  [53] = {x=-3E-06, y=-7.778961, rx=0.301785, ry=175.773697, rz=18.532332, fatherId=world[0]}
  [54] = {x=-4E-06, y=-7.925734, rx=0.301782, ry=175.773696, rz=18.532336, fatherId=world[0]}
  [55] = {x=-4E-06, y=-8.072507, rx=0.301779, ry=175.773696, rz=18.532339, fatherId=world[0]}
  [56] = {x=-4E-06, y=-8.21928, rx=0.301775, ry=175.773696, rz=18.532342, fatherId=world[0]}
  [57] = {x=-4E-06, y=-8.366053, rx=0.301772, ry=175.773696, rz=18.532345, fatherId=world[0]}
  [58] = {x=-4E-06, y=-8.512826, rx=0.301769, ry=175.773695, rz=18.532348, fatherId=world[0]}
  [59] = {x=-4E-06, y=-8.659599, rx=0.301766, ry=175.773695, rz=18.532352, fatherId=world[0]}
  [60] = {x=-4E-06, y=-8.806371, rx=0.301763, ry=175.773695, rz=18.532355, fatherId=world[0]}
  [61] = {x=-4E-06, y=-8.953144, rx=0.301759, ry=175.773694, rz=18.532358, fatherId=world[0]}
  [62] = {x=-4E-06, y=-9.099917, rx=0.301756, ry=175.773694, rz=18.532361, fatherId=world[0]}
  [63] = {x=-4E-06, y=-9.24669, rx=0.301753, ry=175.773694, rz=18.532364, fatherId=world[0]}
  [64] = {x=-4E-06, y=-9.393463, rx=0.30175, ry=175.773693, rz=18.532368, fatherId=world[0]}
  [65] = {x=-4E-06, y=-9.540236, rx=0.301747, ry=175.773693, rz=18.532371, fatherId=world[0]}
  [66] = {x=-4E-06, y=-9.687009, rx=0.301743, ry=175.773693, rz=18.532374, fatherId=world[0]}
  [67] = {x=-4E-06, y=-9.833781, rx=0.30174, ry=175.773693, rz=18.532377, fatherId=world[0]}
  [68] = {x=-5E-06, y=-9.980554, rx=0.301737, ry=175.773692, rz=18.53238, fatherId=world[0]}
  [69] = {x=-5E-06, y=-10.127327, rx=0.301734, ry=175.773692, rz=18.532384, fatherId=world[0]}
  [70] = {x=-5E-06, y=-10.2741, rx=0.301731, ry=175.773692, rz=18.532387, fatherId=world[0]}
  [71] = {x=-5E-06, y=-10.420873, rx=0.301727, ry=175.773692, rz=18.53239, fatherId=world[0]}
  [72] = {x=-5E-06, y=-10.567646, rx=0.301724, ry=175.773691, rz=18.532393, fatherId=world[0]}
  [73] = {x=-5E-06, y=-10.714419, rx=0.301721, ry=175.773691, rz=18.532396, fatherId=world[0]}
  [74] = {x=-5E-06, y=-10.861192, rx=0.301718, ry=175.773691, rz=18.532399, fatherId=world[0]}
  [75] = {x=-5E-06, y=-11.007964, rx=0.301715, ry=175.77369, rz=18.532403, fatherId=world[0]}
  [76] = {x=-5E-06, y=-11.154737, rx=0.301711, ry=175.77369, rz=18.532406, fatherId=world[0]}
  [77] = {x=-5E-06, y=-11.30151, rx=0.301708, ry=175.77369, rz=18.532409, fatherId=world[0]}
  [78] = {x=-5E-06, y=-11.448283, rx=0.301705, ry=175.77369, rz=18.532412, fatherId=world[0]}
  [79] = {x=-5E-06, y=-11.595056, rx=0.301702, ry=175.773689, rz=18.532415, fatherId=world[0]}
  [80] = {x=-5E-06, y=-11.741829, rx=0.301699, ry=175.773689, rz=18.532419, fatherId=world[0]}
  [81] = {x=-5E-06, y=-11.888602, rx=0.301695, ry=175.773689, rz=18.532422, fatherId=world[0]}
  [82] = {x=-6E-06, y=-12.035374, rx=0.301692, ry=175.773688, rz=18.532425, fatherId=world[0]}
  [83] = {x=-6E-06, y=-12.182147, rx=0.301689, ry=175.773688, rz=18.532428, fatherId=world[0]}
  [84] = {x=-6E-06, y=-12.32892, rx=0.301686, ry=175.773688, rz=18.532431, fatherId=world[0]}
  [85] = {x=-6E-06, y=-12.475693, rx=0.301683, ry=175.773688, rz=18.532435, fatherId=world[0]}
  [86] = {x=-6E-06, y=-12.622466, rx=0.301679, ry=175.773687, rz=18.532438, fatherId=world[0]}
  [87] = {x=-6E-06, y=-12.769239, rx=0.301676, ry=175.773687, rz=18.532441, fatherId=world[0]}
  [88] = {x=-6E-06, y=-12.916012, rx=0.301673, ry=175.773687, rz=18.532444, fatherId=world[0]}
  [89] = {x=-6E-06, y=-13.062784, rx=0.30167, ry=175.773687, rz=18.532447, fatherId=world[0]}
  [90] = {x=-6E-06, y=-13.209557, rx=0.301667, ry=175.773686, rz=18.532451, fatherId=world[0]}
  [91] = {x=-6E-06, y=-13.35633, rx=0.301663, ry=175.773686, rz=18.532454, fatherId=world[0]}
  [92] = {x=-6E-06, y=-13.503103, rx=0.30166, ry=175.773686, rz=18.532457, fatherId=world[0]}
  [93] = {x=-6E-06, y=-13.649876, rx=0.301657, ry=175.773685, rz=18.53246, fatherId=world[0]}
  [94] = {x=-6E-06, y=-13.796649, rx=0.301654, ry=175.773685, rz=18.532463, fatherId=world[0]}
  [95] = {x=-7E-06, y=-13.943422, rx=0.301651, ry=175.773685, rz=18.532466, fatherId=world[0]}
  [96] = {x=-7E-06, y=-14.090194, rx=0.301647, ry=175.773685, rz=18.53247, fatherId=world[0]}
  [97] = {x=-7E-06, y=-14.236967, rx=0.301644, ry=175.773684, rz=18.532473, fatherId=world[0]}
  [98] = {x=-7E-06, y=-14.38374, rx=0.301641, ry=175.773684, rz=18.532476, fatherId=world[0]}
  [99] = {x=-7E-06, y=-14.530513, rx=0.301638, ry=175.773684, rz=18.532479, fatherId=world[0]}
  [100] = {x=-7E-06, y=-14.677286, rx=0.301635, ry=175.773684, rz=18.532482, fatherId=world[0]}
  [101] = {x=-7E-06, y=-14.824059, rx=0.301631, ry=175.773683, rz=18.532486, fatherId=world[0]}
  [102] = {x=-7E-06, y=-14.970832, rx=0.301628, ry=175.773683, rz=18.532489, fatherId=world[0]}
  [103] = {x=-7E-06, y=-15.117604, rx=0.301625, ry=175.773683, rz=18.532492, fatherId=world[0]}
  [104] = {x=-7E-06, y=-15.264377, rx=0.301622, ry=175.773683, rz=18.532495, fatherId=world[0]}
  [105] = {x=-7E-06, y=-15.41115, rx=0.301619, ry=175.773682, rz=18.532498, fatherId=world[0]}
  [106] = {x=-7E-06, y=-15.557923, rx=0.301615, ry=175.773682, rz=18.532502, fatherId=world[0]}
  [107] = {x=-7E-06, y=-15.704696, rx=0.301612, ry=175.773682, rz=18.532505, fatherId=world[0]}
  [108] = {x=-8E-06, y=-15.851469, rx=0.301609, ry=175.773681, rz=18.532508, fatherId=world[0]}
  [109] = {x=-8E-06, y=-15.998242, rx=0.301606, ry=175.773681, rz=18.532511, fatherId=world[0]}
  [110] = {x=-8E-06, y=-16.145014, rx=0.301603, ry=175.773681, rz=18.532514, fatherId=world[0]}
  [111] = {x=-8E-06, y=-16.291787, rx=0.301599, ry=175.773681, rz=18.532518, fatherId=world[0]}
  [112] = {x=-8E-06, y=-16.43856, rx=0.301596, ry=175.77368, rz=18.532521, fatherId=world[0]}
  [113] = {x=-8E-06, y=-16.585333, rx=0.301593, ry=175.77368, rz=18.532524, fatherId=world[0]}
  [114] = {x=-8E-06, y=-16.732106, rx=0.30159, ry=175.77368, rz=18.532527, fatherId=world[0]}
  [115] = {x=-8E-06, y=-16.878879, rx=0.301587, ry=175.77368, rz=18.53253, fatherId=world[0]}
  [116] = {x=-8E-06, y=-17.025652, rx=0.301583, ry=175.773679, rz=18.532534, fatherId=world[0]}
  [117] = {x=-8E-06, y=-17.172424, rx=0.30158, ry=175.773679, rz=18.532537, fatherId=world[0]}
  [118] = {x=-8E-06, y=-17.319197, rx=0.301577, ry=175.773679, rz=18.53254, fatherId=world[0]}
  [119] = {x=-8E-06, y=-17.46597, rx=0.301574, ry=175.773679, rz=18.532543, fatherId=world[0]}
  [120] = {x=-8E-06, y=-17.612743, rx=0.301571, ry=175.773678, rz=18.532546, fatherId=world[0]}
  [121] = {x=-9E-06, y=-17.759516, rx=0.301567, ry=175.773678, rz=18.53255, fatherId=world[0]}
  [122] = {x=-9E-06, y=-17.906289, rx=0.301564, ry=175.773678, rz=18.532553, fatherId=world[0]}
  [123] = {x=-9E-06, y=-18.053062, rx=0.301561, ry=175.773678, rz=18.532556, fatherId=world[0]}
  [124] = {x=-9E-06, y=-18.199834, rx=0.301558, ry=175.773677, rz=18.532559, fatherId=world[0]}
  [125] = {x=-9E-06, y=-18.346607, rx=0.301555, ry=175.773677, rz=18.532562, fatherId=world[0]}
  [126] = {x=-9E-06, y=-18.49338, rx=0.301551, ry=175.773677, rz=18.532566, fatherId=world[0]}
  [127] = {x=-9E-06, y=-18.640153, rx=0.301548, ry=175.773677, rz=18.532569, fatherId=world[0]}
  [128] = {x=-9E-06, y=-18.786926, rx=0.301545, ry=175.773676, rz=18.532572, fatherId=world[0]}
  [129] = {x=-9E-06, y=-18.933699, rx=0.301542, ry=175.773676, rz=18.532575, fatherId=world[0]}
  [130] = {x=-9E-06, y=-19.080472, rx=0.301538, ry=175.773676, rz=18.532578, fatherId=world[0]}
  [131] = {x=-9E-06, y=-19.227244, rx=0.301535, ry=175.773676, rz=18.532582, fatherId=world[0]}
  [132] = {x=-9E-06, y=-19.374017, rx=0.301532, ry=175.773675, rz=18.532585, fatherId=world[0]}
  [133] = {x=-1E-05, y=-19.52079, z=-1E-06, rx=0.301529, ry=175.773675, rz=18.532588, fatherId=world[0]}
  [134] = {x=-1E-05, y=-19.667563, z=-1E-06, rx=0.301526, ry=175.773675, rz=18.532591, fatherId=world[0]}
  [135] = {x=-1E-05, y=-19.814336, z=-1E-06, rx=0.301522, ry=175.773675, rz=18.532594, fatherId=world[0]}
  [136] = {x=-1E-05, y=-19.961109, z=-1E-06, rx=0.301519, ry=175.773674, rz=18.532598, fatherId=world[0]}
  [137] = {x=-1E-05, y=-20.107882, z=-1E-06, rx=0.301516, ry=175.773674, rz=18.532601, fatherId=world[0]}
  [138] = {x=-1E-05, y=-20.254654, z=-1E-06, rx=0.301513, ry=175.773674, rz=18.532604, fatherId=world[0]}
  [139] = {x=-1E-05, y=-20.401427, z=-1E-06, rx=0.30151, ry=175.773674, rz=18.532607, fatherId=world[0]}
  [140] = {x=-1E-05, y=-20.5482, z=-1E-06, rx=0.301506, ry=175.773673, rz=18.53261, fatherId=world[0]}
  [141] = {x=-1E-05, y=-20.694973, z=-1E-06, rx=0.301503, ry=175.773673, rz=18.532614, fatherId=world[0]}
  [142] = {x=-1E-05, y=-20.841746, z=-1E-06, rx=0.3015, ry=175.773673, rz=18.532617, fatherId=world[0]}
  [143] = {x=-1E-05, y=-20.988519, z=-1E-06, rx=0.301497, ry=175.773673, rz=18.53262, fatherId=world[0]}
  [144] = {x=-1E-05, y=-21.135292, z=-1E-06, rx=0.301494, ry=175.773673, rz=18.532623, fatherId=world[0]}
  [145] = {x=-1E-05, y=-21.282064, z=-1E-06, rx=0.30149, ry=175.773672, rz=18.532626, fatherId=world[0]}
  [146] = {x=-1.1E-05, y=-21.428837, z=-1E-06, rx=0.301487, ry=175.773672, rz=18.53263, fatherId=world[0]}
  [147] = {x=-1.1E-05, y=-21.57561, z=-1E-06, rx=0.301484, ry=175.773672, rz=18.532633, fatherId=world[0]}
  [148] = {x=-1.1E-05, y=-21.722383, z=-1E-06, rx=0.301481, ry=175.773672, rz=18.532636, fatherId=world[0]}
  [149] = {x=-1.1E-05, y=-21.869156, z=-1E-06, rx=0.301477, ry=175.773671, rz=18.532639, fatherId=world[0]}
  [150] = {x=-1.1E-05, y=-22.015929, z=-1E-06, rx=0.301474, ry=175.773671, rz=18.532642, fatherId=world[0]}
  [151] = {x=-1.1E-05, y=-22.162702, z=-1E-06, rx=0.301471, ry=175.773671, rz=18.532646, fatherId=world[0]}
  [152] = {x=-1.1E-05, y=-22.309474, z=-1E-06, rx=0.301468, ry=175.773671, rz=18.532649, fatherId=world[0]}
  [153] = {x=-1.1E-05, y=-22.456247, z=-1E-06, rx=0.301465, ry=175.77367, rz=18.532652, fatherId=world[0]}
  [154] = {x=-1.1E-05, y=-22.60302, z=-1E-06, rx=0.301461, ry=175.77367, rz=18.532655, fatherId=world[0]}
  [155] = {x=-1.1E-05, y=-22.749793, z=-1E-06, rx=0.301458, ry=175.77367, rz=18.532658, fatherId=world[0]}
  [156] = {x=-1.1E-05, y=-22.896566, z=-1E-06, rx=0.301455, ry=175.77367, rz=18.532662, fatherId=world[0]}
  [157] = {x=-1.1E-05, y=-23.043339, z=-1E-06, rx=0.301452, ry=175.773669, rz=18.532665, fatherId=world[0]}
  [158] = {x=-1.2E-05, y=-23.190112, z=-1E-06, rx=0.301449, ry=175.773669, rz=18.532668, fatherId=world[0]}
  [159] = {x=-1.2E-05, y=-23.336884, z=-1E-06, rx=0.301445, ry=175.773669, rz=18.532671, fatherId=world[0]}
  [160] = {x=-1.2E-05, y=-23.483657, z=-1E-06, rx=0.301442, ry=175.773669, rz=18.532674, fatherId=world[0]}
  [161] = {x=-1.2E-05, y=-23.63043, z=-1E-06, rx=0.301439, ry=175.773669, rz=18.532678, fatherId=world[0]}
  [162] = {x=-1.2E-05, y=-23.777203, z=-1E-06, rx=0.301436, ry=175.773668, rz=18.532681, fatherId=world[0]}
  [163] = {x=-1.2E-05, y=-23.923976, z=-1E-06, rx=0.301433, ry=175.773668, rz=18.532684, fatherId=world[0]}
  [164] = {x=-1.2E-05, y=-24.070749, z=-1E-06, rx=0.301429, ry=175.773668, rz=18.532687, fatherId=world[0]}
  [165] = {x=-1.2E-05, y=-24.217522, z=-1E-06, rx=0.301426, ry=175.773668, rz=18.53269, fatherId=world[0]}
  [166] = {x=-1.2E-05, y=-24.364294, z=-1E-06, rx=0.301423, ry=175.773667, rz=18.532694, fatherId=world[0]}
  [167] = {x=-1.2E-05, y=-24.511067, z=-1E-06, rx=0.30142, ry=175.773667, rz=18.532697, fatherId=world[0]}
  [168] = {x=-1.2E-05, y=-24.65784, z=-1E-06, rx=0.301416, ry=175.773667, rz=18.5327, fatherId=world[0]}
  [169] = {x=-1.3E-05, y=-24.804613, z=-1E-06, rx=0.301413, ry=175.773667, rz=18.532703, fatherId=world[0]}
  [170] = {x=-1.3E-05, y=-24.951386, z=-1E-06, rx=0.30141, ry=175.773667, rz=18.532706, fatherId=world[0]}
  [171] = {x=-1.3E-05, y=-25.098159, z=-1E-06, rx=0.301407, ry=175.773666, rz=18.53271, fatherId=world[0]}
  [172] = {x=-1.3E-05, y=-25.244932, z=-1E-06, rx=0.301404, ry=175.773666, rz=18.532713, fatherId=world[0]}
  [173] = {x=-1.3E-05, y=-25.391704, z=-1E-06, rx=0.3014, ry=175.773666, rz=18.532716, fatherId=world[0]}
  [174] = {x=-1.3E-05, y=-25.538477, z=-1E-06, rx=0.301397, ry=175.773666, rz=18.532719, fatherId=world[0]}
  [175] = {x=-1.3E-05, y=-25.68525, z=-1E-06, rx=0.301394, ry=175.773665, rz=18.532722, fatherId=world[0]}
  [176] = {x=-1.3E-05, y=-25.832023, z=-1E-06, rx=0.301391, ry=175.773665, rz=18.532726, fatherId=world[0]}
  [177] = {x=-1.3E-05, y=-25.978796, z=-1E-06, rx=0.301388, ry=175.773665, rz=18.532729, fatherId=world[0]}
  [178] = {x=-1.3E-05, y=-26.125569, z=-1E-06, rx=0.301384, ry=175.773665, rz=18.532732, fatherId=world[0]}
  [179] = {x=-1.3E-05, y=-26.272342, z=-1E-06, rx=0.301381, ry=175.773665, rz=18.532735, fatherId=world[0]}
  [180] = {x=-1.3E-05, y=-26.419114, z=-1E-06, rx=0.301378, ry=175.773664, rz=18.532738, fatherId=world[0]}
  [181] = {x=-1.4E-05, y=-26.565887, z=-1E-06, rx=0.301375, ry=175.773664, rz=18.532742, fatherId=world[0]}
  [182] = {x=-1.4E-05, y=-26.71266, z=-1E-06, rx=0.301371, ry=175.773664, rz=18.532745, fatherId=world[0]}
  [183] = {x=-1.4E-05, y=-26.859433, z=-1E-06, rx=0.301368, ry=175.773664, rz=18.532748, fatherId=world[0]}
  [184] = {x=-1.4E-05, y=-27.006206, z=-1E-06, rx=0.301365, ry=175.773664, rz=18.532751, fatherId=world[0]}
  [185] = {x=-1.4E-05, y=-27.152979, z=-1E-06, rx=0.301362, ry=175.773663, rz=18.532754, fatherId=world[0]}
  [186] = {x=-1.4E-05, y=-27.299752, z=-1E-06, rx=0.301359, ry=175.773663, rz=18.532758, fatherId=world[0]}
  [187] = {x=-1.4E-05, y=-27.446524, z=-1E-06, rx=0.301355, ry=175.773663, rz=18.532761, fatherId=world[0]}
  [188] = {x=-1.4E-05, y=-27.593297, z=-1E-06, rx=0.301352, ry=175.773663, rz=18.532764, fatherId=world[0]}
  [189] = {x=-1.4E-05, y=-27.74007, z=-1E-06, rx=0.301349, ry=175.773662, rz=18.532767, fatherId=world[0]}
  [190] = {x=-1.4E-05, y=-27.886843, z=-1E-06, rx=0.301346, ry=175.773662, rz=18.53277, fatherId=world[0]}
  [191] = {x=-1.4E-05, y=-28.033616, z=-1E-06, rx=0.301343, ry=175.773662, rz=18.532774, fatherId=world[0]}
  [192] = {x=-1.5E-05, y=-28.180389, z=-1E-06, rx=0.301339, ry=175.773662, rz=18.532777, fatherId=world[0]}
  [193] = {x=-1.5E-05, y=-28.327162, z=-1E-06, rx=0.301336, ry=175.773662, rz=18.53278, fatherId=world[0]}
  [194] = {x=-1.5E-05, y=-28.473934, z=-1E-06, rx=0.301333, ry=175.773661, rz=18.532783, fatherId=world[0]}
  [195] = {x=-1.5E-05, y=-28.620707, z=-1E-06, rx=0.30133, ry=175.773661, rz=18.532786, fatherId=world[0]}
  [196] = {x=-1.5E-05, y=-28.76748, z=-1E-06, rx=0.301326, ry=175.773661, rz=18.53279, fatherId=world[0]}
  [197] = {x=-1.5E-05, y=-28.914253, z=-1E-06, rx=0.301323, ry=175.773661, rz=18.532793, fatherId=world[0]}
  [198] = {x=-1.5E-05, y=-29.061026, z=-1E-06, rx=0.30132, ry=175.773661, rz=18.532796, fatherId=world[0]}
  [199] = {x=-1.5E-05, y=-29.207799, z=-1E-06, rx=0.301317, ry=175.77366, rz=18.532799, fatherId=world[0]}
  [200] = {x=-1.5E-05, y=-29.354572, z=-1E-06, rx=0.301314, ry=175.77366, rz=18.532802, fatherId=world[0]}
  [201] = {x=-1.5E-05, y=-29.501344, z=-1E-06, rx=0.30131, ry=175.77366, rz=18.532806, fatherId=world[0]}
  [202] = {x=-1.5E-05, y=-29.648117, z=-1E-06, rx=0.301307, ry=175.77366, rz=18.532809, fatherId=world[0]}
  [203] = {x=-1.6E-05, y=-29.79489, z=-1E-06, rx=0.301304, ry=175.77366, rz=18.532812, fatherId=world[0]}
  [204] = {x=-1.6E-05, y=-29.941663, z=-1E-06, rx=0.301301, ry=175.773659, rz=18.532815, fatherId=world[0]}
  [205] = {x=-1.6E-05, y=-30.088436, z=-1E-06, rx=0.301297, ry=175.773659, rz=18.532819, fatherId=world[0]}
  [206] = {x=-1.6E-05, y=-30.235209, z=-1E-06, rx=0.301294, ry=175.773659, rz=18.532822, fatherId=world[0]}
  [207] = {x=-1.6E-05, y=-30.381982, z=-1E-06, rx=0.301291, ry=175.773659, rz=18.532825, fatherId=world[0]}
  [208] = {x=-1.6E-05, y=-30.528755, z=-1E-06, rx=0.301288, ry=175.773659, rz=18.532828, fatherId=world[0]}
  [209] = {x=-1.6E-05, y=-30.675527, z=-1E-06, rx=0.301285, ry=175.773658, rz=18.532831, fatherId=world[0]}
  [210] = {x=-1.6E-05, y=-30.8223, z=-1E-06, rx=0.301281, ry=175.773658, rz=18.532835, fatherId=world[0]}
  [211] = {x=-1.6E-05, y=-30.969073, z=-1E-06, rx=0.301278, ry=175.773658, rz=18.532838, fatherId=world[0]}
  [212] = {x=-1.6E-05, y=-31.115846, z=-1E-06, rx=0.301275, ry=175.773658, rz=18.532841, fatherId=world[0]}
  [213] = {x=-1.6E-05, y=-31.262619, z=-1E-06, rx=0.301272, ry=175.773658, rz=18.532844, fatherId=world[0]}
  [214] = {x=-1.7E-05, y=-31.409392, z=-1E-06, rx=0.301269, ry=175.773657, rz=18.532847, fatherId=world[0]}
  [215] = {x=-1.7E-05, y=-31.556165, z=-1E-06, rx=0.301265, ry=175.773657, rz=18.532851, fatherId=world[0]}
  [216] = {x=-1.7E-05, y=-31.702937, z=-1E-06, rx=0.301262, ry=175.773657, rz=18.532854, fatherId=world[0]}
  [217] = {x=-1.7E-05, y=-31.84971, z=-1E-06, rx=0.301259, ry=175.773657, rz=18.532857, fatherId=world[0]}
  [218] = {x=-1.7E-05, y=-31.996483, z=-1E-06, rx=0.301256, ry=175.773657, rz=18.53286, fatherId=world[0]}
  [219] = {x=-1.7E-05, y=-32.143256, z=-1E-06, rx=0.301252, ry=175.773656, rz=18.532863, fatherId=world[0]}
  [220] = {x=-1.7E-05, y=-32.290029, z=-1E-06, rx=0.301249, ry=175.773656, rz=18.532867, fatherId=world[0]}
  [221] = {x=-1.7E-05, y=-32.436802, z=-1E-06, rx=0.301246, ry=175.773656, rz=18.53287, fatherId=world[0]}
  [222] = {x=-1.7E-05, y=-32.583575, z=-1E-06, rx=0.301243, ry=175.773656, rz=18.532873, fatherId=world[0]}
  [223] = {x=-1.7E-05, y=-32.730347, z=-1E-06, rx=0.30124, ry=175.773656, rz=18.532876, fatherId=world[0]}
  [224] = {x=-1.7E-05, y=-32.87712, z=-1E-06, rx=0.301236, ry=175.773656, rz=18.532879, fatherId=world[0]}
  [225] = {x=-1.8E-05, y=-33.023893, z=-1E-06, rx=0.301233, ry=175.773655, rz=18.532883, fatherId=world[0]}
  [226] = {x=-1.8E-05, y=-33.170666, z=-1E-06, rx=0.30123, ry=175.773655, rz=18.532886, fatherId=world[0]}
  [227] = {x=-1.8E-05, y=-33.317439, z=-1E-06, rx=0.301227, ry=175.773655, rz=18.532889, fatherId=world[0]}
  [228] = {x=-1.8E-05, y=-33.464212, z=-1E-06, rx=0.301223, ry=175.773655, rz=18.532892, fatherId=world[0]}
  [229] = {x=-1.8E-05, y=-33.610985, z=-1E-06, rx=0.30122, ry=175.773655, rz=18.532896, fatherId=world[0]}
  [230] = {x=-1.8E-05, y=-33.757757, z=-1E-06, rx=0.301217, ry=175.773654, rz=18.532899, fatherId=world[0]}
  [231] = {x=-1.8E-05, y=-33.90453, z=-1E-06, rx=0.301214, ry=175.773654, rz=18.532902, fatherId=world[0]}
  [232] = {x=-1.8E-05, y=-34.051303, z=-1E-06, rx=0.301211, ry=175.773654, rz=18.532905, fatherId=world[0]}
  [233] = {x=-1.8E-05, y=-34.198076, z=-1E-06, rx=0.301207, ry=175.773654, rz=18.532908, fatherId=world[0]}
  [234] = {x=-1.8E-05, y=-34.344849, z=-1E-06, rx=0.301204, ry=175.773654, rz=18.532912, fatherId=world[0]}
  [235] = {x=-1.9E-05, y=-34.491622, z=-1E-06, rx=0.301201, ry=175.773654, rz=18.532915, fatherId=world[0]}
  [236] = {x=-1.9E-05, y=-34.638395, z=-1E-06, rx=0.301198, ry=175.773653, rz=18.532918, fatherId=world[0]}
  [237] = {x=-1.9E-05, y=-34.785167, z=-1E-06, rx=0.301194, ry=175.773653, rz=18.532921, fatherId=world[0]}
  [238] = {x=-1.9E-05, y=-34.93194, z=-1E-06, rx=0.301191, ry=175.773653, rz=18.532924, fatherId=world[0]}
  [239] = {x=-1.9E-05, y=-35.078713, z=-1E-06, rx=0.301188, ry=175.773653, rz=18.532928, fatherId=world[0]}
  [240] = {x=-1.9E-05, y=-35.225486, z=-1E-06, rx=0.301185, ry=175.773653, rz=18.532931, fatherId=world[0]}
  [241] = {x=-1.9E-05, y=-35.372259, z=-1E-06, rx=0.301182, ry=175.773652, rz=18.532934, fatherId=world[0]}
  [242] = {x=-1.9E-05, y=-35.519032, z=-1E-06, rx=0.301178, ry=175.773652, rz=18.532937, fatherId=world[0]}
  [243] = {x=-1.9E-05, y=-35.665805, z=-1E-06, rx=0.301175, ry=175.773652, rz=18.53294, fatherId=world[0]}
  [244] = {x=-1.9E-05, y=-35.812577, z=-1E-06, rx=0.301172, ry=175.773652, rz=18.532944, fatherId=world[0]}
  [245] = {x=-1.9E-05, y=-35.95935, z=-1E-06, rx=0.301169, ry=175.773652, rz=18.532947, fatherId=world[0]}
  [246] = {x=-2E-05, y=-36.106123, z=-1E-06, rx=0.301165, ry=175.773652, rz=18.53295, fatherId=world[0]}
  [247] = {x=-2E-05, y=-36.252896, z=-1E-06, rx=0.301162, ry=175.773651, rz=18.532953, fatherId=world[0]}
  [248] = {x=-2E-05, y=-36.399669, z=-1E-06, rx=0.301159, ry=175.773651, rz=18.532957, fatherId=world[0]}
  [249] = {x=-2E-05, y=-36.546442, z=-1E-06, rx=0.301156, ry=175.773651, rz=18.53296, fatherId=world[0]}
  [250] = {x=-2E-05, y=-36.693215, z=-1E-06, rx=0.301153, ry=175.773651, rz=18.532963, fatherId=world[0]}
  [251] = {x=-2E-05, y=-36.839987, z=-1E-06, rx=0.301149, ry=175.773651, rz=18.532966, fatherId=world[0]}
  [252] = {x=-2E-05, y=-36.98676, z=-1E-06, rx=0.301146, ry=175.773651, rz=18.532969, fatherId=world[0]}
  [253] = {x=-2E-05, y=-37.133533, z=-1E-06, rx=0.301143, ry=175.77365, rz=18.532973, fatherId=world[0]}
  [254] = {x=-2E-05, y=-37.280306, z=-1E-06, rx=0.30114, ry=175.77365, rz=18.532976, fatherId=world[0]}
  [255] = {x=-2E-05, y=-37.427079, z=-1E-06, rx=0.301136, ry=175.77365, rz=18.532979, fatherId=world[0]}
  [256] = {x=-2.1E-05, y=-37.573852, z=-1E-06, rx=0.301133, ry=175.77365, rz=18.532982, fatherId=world[0]}
  [257] = {x=-2.1E-05, y=-37.720625, z=-1E-06, rx=0.30113, ry=175.77365, rz=18.532985, fatherId=world[0]}
  [258] = {x=-2.1E-05, y=-37.867397, z=-1E-06, rx=0.301127, ry=175.77365, rz=18.532989, fatherId=world[0]}
  [259] = {x=-2.1E-05, y=-38.01417, z=-1E-06, rx=0.301123, ry=175.773649, rz=18.532992, fatherId=world[0]}
  [260] = {x=-2.1E-05, y=-38.160943, z=-1E-06, rx=0.30112, ry=175.773649, rz=18.532995, fatherId=world[0]}
  [261] = {x=-2.1E-05, y=-38.307716, z=-1E-06, rx=0.301117, ry=175.773649, rz=18.532998, fatherId=world[0]}
  [262] = {x=-2.1E-05, y=-38.454489, z=-1E-06, rx=0.301114, ry=175.773649, rz=18.533002, fatherId=world[0]}
  [263] = {x=-2.1E-05, y=-38.601262, z=-1E-06, rx=0.301111, ry=175.773649, rz=18.533005, fatherId=world[0]}
  [264] = {x=-2.1E-05, y=-38.748035, z=-1E-06, rx=0.301107, ry=175.773649, rz=18.533008, fatherId=world[0]}
  [265] = {x=-2.1E-05, y=-38.894807, z=-1E-06, rx=0.301104, ry=175.773648, rz=18.533011, fatherId=world[0]}
  [266] = {x=-2.2E-05, y=-39.04158, z=-1E-06, rx=0.301101, ry=175.773648, rz=18.533014, fatherId=world[0]}
  [267] = {x=-2.2E-05, y=-39.188353, z=-1E-06, rx=0.301098, ry=175.773648, rz=18.533018, fatherId=world[0]}
  [268] = {x=-2.2E-05, y=-39.335126, z=-1E-06, rx=0.301094, ry=175.773648, rz=18.533021, fatherId=world[0]}
  [269] = {x=-2.2E-05, y=-39.481899, z=-1E-06, rx=0.301091, ry=175.773648, rz=18.533024, fatherId=world[0]}
  [270] = {x=-2.2E-05, y=-39.628672, z=-2E-06, rx=0.301088, ry=175.773648, rz=18.533027, fatherId=world[0]}
  [271] = {x=-2.2E-05, y=-39.775445, z=-2E-06, rx=0.301085, ry=175.773647, rz=18.53303, fatherId=world[0]}
  [272] = {x=-2.2E-05, y=-39.922217, z=-2E-06, rx=0.301082, ry=175.773647, rz=18.533034, fatherId=world[0]}
  [273] = {x=-2.2E-05, y=-40.06899, z=-2E-06, rx=0.301078, ry=175.773647, rz=18.533037, fatherId=world[0]}
  [274] = {x=-2.2E-05, y=-40.215763, z=-2E-06, rx=0.301075, ry=175.773647, rz=18.53304, fatherId=world[0]}
  [275] = {x=-2.2E-05, y=-40.362536, z=-2E-06, rx=0.301072, ry=175.773647, rz=18.533043, fatherId=world[0]}
  [276] = {x=-2.3E-05, y=-40.509309, z=-2E-06, rx=0.301069, ry=175.773647, rz=18.533047, fatherId=world[0]}
  [277] = {x=-2.3E-05, y=-40.656082, z=-2E-06, rx=0.301065, ry=175.773646, rz=18.53305, fatherId=world[0]}
  [278] = {x=-2.3E-05, y=-40.802855, z=-2E-06, rx=0.301062, ry=175.773646, rz=18.533053, fatherId=world[0]}
  [279] = {x=-2.3E-05, y=-40.949627, z=-2E-06, rx=0.301059, ry=175.773646, rz=18.533056, fatherId=world[0]}
  [280] = {x=-2.3E-05, y=-41.0964, z=-2E-06, rx=0.301056, ry=175.773646, rz=18.533059, fatherId=world[0]}
  [281] = {x=-2.3E-05, y=-41.243173, z=-2E-06, rx=0.301052, ry=175.773646, rz=18.533063, fatherId=world[0]}
  [282] = {x=-2.3E-05, y=-41.389946, z=-2E-06, rx=0.301049, ry=175.773646, rz=18.533066, fatherId=world[0]}
  [283] = {x=-2.3E-05, y=-41.536719, z=-2E-06, rx=0.301046, ry=175.773646, rz=18.533069, fatherId=world[0]}
  [284] = {x=-2.3E-05, y=-41.683492, z=-2E-06, rx=0.301043, ry=175.773645, rz=18.533072, fatherId=world[0]}
  [285] = {x=-2.3E-05, y=-41.830265, z=-2E-06, rx=0.30104, ry=175.773645, rz=18.533075, fatherId=world[0]}
  [286] = {x=-2.4E-05, y=-41.977037, z=-2E-06, rx=0.301036, ry=175.773645, rz=18.533079, fatherId=world[0]}
  [287] = {x=-2.4E-05, y=-42.12381, z=-2E-06, rx=0.301033, ry=175.773645, rz=18.533082, fatherId=world[0]}
  [288] = {x=-2.4E-05, y=-42.270583, z=-2E-06, rx=0.30103, ry=175.773645, rz=18.533085, fatherId=world[0]}
  [289] = {x=-2.4E-05, y=-42.417356, z=-2E-06, rx=0.301027, ry=175.773645, rz=18.533088, fatherId=world[0]}
  [290] = {x=-2.4E-05, y=-42.564129, z=-2E-06, rx=0.301023, ry=175.773645, rz=18.533092, fatherId=world[0]}
  [291] = {x=-2.4E-05, y=-42.710902, z=-2E-06, rx=0.30102, ry=175.773644, rz=18.533095, fatherId=world[0]}
  [292] = {x=-2.4E-05, y=-42.857675, z=-2E-06, rx=0.301017, ry=175.773644, rz=18.533098, fatherId=world[0]}
  [293] = {x=-2.4E-05, y=-43.004447, z=-2E-06, rx=0.301014, ry=175.773644, rz=18.533101, fatherId=world[0]}
  [294] = {x=-2.4E-05, y=-43.15122, z=-2E-06, rx=0.30101, ry=175.773644, rz=18.533104, fatherId=world[0]}
  [295] = {x=-2.4E-05, y=-43.297993, z=-2E-06, rx=0.301007, ry=175.773644, rz=18.533108, fatherId=world[0]}
  [296] = {x=-2.5E-05, y=-43.444766, z=-2E-06, rx=0.301004, ry=175.773644, rz=18.533111, fatherId=world[0]}
  [297] = {x=-2.5E-05, y=-43.591539, z=-2E-06, rx=0.301001, ry=175.773644, rz=18.533114, fatherId=world[0]}
  [298] = {x=-2.5E-05, y=-43.738312, z=-2E-06, rx=0.300998, ry=175.773643, rz=18.533117, fatherId=world[0]}
  [299] = {x=-2.5E-05, y=-43.885085, z=-2E-06, rx=0.300994, ry=175.773643, rz=18.533121, fatherId=world[0]}
  [300] = {x=-2.5E-05, y=-44.031857, z=-2E-06, rx=0.300991, ry=175.773643, rz=18.533124, fatherId=world[0]}
  [301] = {x=-2.5E-05, y=-44.17863, z=-2E-06, rx=0.300988, ry=175.773643, rz=18.533127, fatherId=world[0]}
  [302] = {x=-2.5E-05, y=-44.325403, z=-2E-06, rx=0.300985, ry=175.773643, rz=18.53313, fatherId=world[0]}
  [303] = {x=-2.5E-05, y=-44.472176, z=-2E-06, rx=0.300981, ry=175.773643, rz=18.533133, fatherId=world[0]}
  [304] = {x=-2.5E-05, y=-44.618949, z=-2E-06, rx=0.300978, ry=175.773643, rz=18.533137, fatherId=world[0]}
  [305] = {x=-2.6E-05, y=-44.765722, z=-2E-06, rx=0.300975, ry=175.773642, rz=18.53314, fatherId=world[0]}
  [306] = {x=-2.6E-05, y=-44.912495, z=-2E-06, rx=0.300972, ry=175.773642, rz=18.533143, fatherId=world[0]}
  [307] = {x=-2.6E-05, y=-45.059267, z=-2E-06, rx=0.300968, ry=175.773642, rz=18.533146, fatherId=world[0]}
  [308] = {x=-2.6E-05, y=-45.20604, z=-2E-06, rx=0.300965, ry=175.773642, rz=18.533149, fatherId=world[0]}
  [309] = {x=-2.6E-05, y=-45.352813, z=-2E-06, rx=0.300962, ry=175.773642, rz=18.533153, fatherId=world[0]}
  [310] = {x=-2.6E-05, y=-45.499586, z=-2E-06, rx=0.300959, ry=175.773642, rz=18.533156, fatherId=world[0]}
  [311] = {x=-2.6E-05, y=-45.646359, z=-2E-06, rx=0.300956, ry=175.773642, rz=18.533159, fatherId=world[0]}
  [312] = {x=-2.6E-05, y=-45.793132, z=-2E-06, rx=0.300952, ry=175.773641, rz=18.533162, fatherId=world[0]}
  [313] = {x=-2.6E-05, y=-45.939905, z=-2E-06, rx=0.300949, ry=175.773641, rz=18.533166, fatherId=world[0]}
  [314] = {x=-2.7E-05, y=-46.086677, z=-2E-06, rx=0.300946, ry=175.773641, rz=18.533169, fatherId=world[0]}
  [315] = {x=-2.7E-05, y=-46.23345, z=-2E-06, rx=0.300943, ry=175.773641, rz=18.533172, fatherId=world[0]}
  [316] = {x=-2.7E-05, y=-46.380223, z=-2E-06, rx=0.300939, ry=175.773641, rz=18.533175, fatherId=world[0]}
  [317] = {x=-2.7E-05, y=-46.526996, z=-2E-06, rx=0.300936, ry=175.773641, rz=18.533178, fatherId=world[0]}
  [318] = {x=-2.7E-05, y=-46.673769, z=-2E-06, rx=0.300933, ry=175.773641, rz=18.533182, fatherId=world[0]}
  [319] = {x=-2.7E-05, y=-46.820542, z=-2E-06, rx=0.30093, ry=175.773641, rz=18.533185, fatherId=world[0]}
  [320] = {x=-2.7E-05, y=-46.967315, z=-2E-06, rx=0.300926, ry=175.77364, rz=18.533188, fatherId=world[0]}
  [321] = {x=-2.7E-05, y=-47.114088, z=-2E-06, rx=0.300923, ry=175.77364, rz=18.533191, fatherId=world[0]}
  [322] = {x=-2.7E-05, y=-47.26086, z=-2E-06, rx=0.30092, ry=175.77364, rz=18.533195, fatherId=world[0]}
  [323] = {x=-2.7E-05, y=-47.407633, z=-2E-06, rx=0.300917, ry=175.77364, rz=18.533198, fatherId=world[0]}
  [324] = {x=-2.8E-05, y=-47.554406, z=-2E-06, rx=0.300914, ry=175.77364, rz=18.533201, fatherId=world[0]}
  [325] = {x=-2.8E-05, y=-47.701179, z=-2E-06, rx=0.30091, ry=175.77364, rz=18.533204, fatherId=world[0]}
  [326] = {x=-2.8E-05, y=-47.847952, z=-2E-06, rx=0.300907, ry=175.77364, rz=18.533207, fatherId=world[0]}
  [327] = {x=-2.8E-05, y=-47.994725, z=-2E-06, rx=0.300904, ry=175.77364, rz=18.533211, fatherId=world[0]}
  [328] = {x=-2.8E-05, y=-48.141498, z=-2E-06, rx=0.300901, ry=175.773639, rz=18.533214, fatherId=world[0]}
  [329] = {x=-2.8E-05, y=-48.28827, z=-2E-06, rx=0.300897, ry=175.773639, rz=18.533217, fatherId=world[0]}
  [330] = {x=-2.8E-05, y=-48.435043, z=-2E-06, rx=0.300894, ry=175.773639, rz=18.53322, fatherId=world[0]}
  [331] = {x=-2.8E-05, y=-48.581816, z=-2E-06, rx=0.300891, ry=175.773639, rz=18.533224, fatherId=world[0]}
  [332] = {x=-2.8E-05, y=-48.728589, z=-2E-06, rx=0.300888, ry=175.773639, rz=18.533227, fatherId=world[0]}
  [333] = {x=-2.9E-05, y=-48.875362, z=-2E-06, rx=0.300884, ry=175.773639, rz=18.53323, fatherId=world[0]}
  [334] = {x=-2.9E-05, y=-49.022135, z=-2E-06, rx=0.300881, ry=175.773639, rz=18.533233, fatherId=world[0]}
  [335] = {x=-2.9E-05, y=-49.168908, z=-2E-06, rx=0.300878, ry=175.773639, rz=18.533236, fatherId=world[0]}
  [336] = {x=-2.9E-05, y=-49.31568, z=-2E-06, rx=0.300875, ry=175.773638, rz=18.53324, fatherId=world[0]}
  [337] = {x=-2.9E-05, y=-49.462453, z=-2E-06, rx=0.300871, ry=175.773638, rz=18.533243, fatherId=world[0]}
  [338] = {x=-2.9E-05, y=-49.609226, z=-2E-06, rx=0.300868, ry=175.773638, rz=18.533246, fatherId=world[0]}
  [339] = {x=-2.9E-05, y=-49.755999, z=-2E-06, rx=0.300865, ry=175.773638, rz=18.533249, fatherId=world[0]}
  [340] = {x=-2.9E-05, y=-49.902772, z=-2E-06, rx=0.300862, ry=175.773638, rz=18.533253, fatherId=world[0]}
  [341] = {x=-2.9E-05, y=-50.049545, z=-2E-06, rx=0.300858, ry=175.773638, rz=18.533256, fatherId=world[0]}
  [342] = {x=-3E-05, y=-50.196318, z=-2E-06, rx=0.300855, ry=175.773638, rz=18.533259, fatherId=world[0]}
  [343] = {x=-3E-05, y=-50.34309, z=-2E-06, rx=0.300852, ry=175.773638, rz=18.533262, fatherId=world[0]}
  [344] = {x=-3E-05, y=-50.489863, z=-2E-06, rx=0.300849, ry=175.773638, rz=18.533265, fatherId=world[0]}
  [345] = {x=-3E-05, y=-50.636636, z=-2E-06, rx=0.300846, ry=175.773637, rz=18.533269, fatherId=world[0]}
  [346] = {x=-3E-05, y=-50.783409, z=-2E-06, rx=0.300842, ry=175.773637, rz=18.533272, fatherId=world[0]}
  [347] = {x=-3E-05, y=-50.930182, z=-2E-06, rx=0.300839, ry=175.773637, rz=18.533275, fatherId=world[0]}
  [348] = {x=-3E-05, y=-51.076955, z=-2E-06, rx=0.300836, ry=175.773637, rz=18.533278, fatherId=world[0]}
  [349] = {x=-3E-05, y=-51.223728, z=-2E-06, rx=0.300833, ry=175.773637, rz=18.533282, fatherId=world[0]}
  [350] = {x=-3E-05, y=-51.3705, z=-2E-06, rx=0.300829, ry=175.773637, rz=18.533285, fatherId=world[0]}
  [351] = {x=-3.1E-05, y=-51.517273, z=-2E-06, rx=0.300826, ry=175.773637, rz=18.533288, fatherId=world[0]}
  [352] = {x=-3.1E-05, y=-51.664046, z=-2E-06, rx=0.300823, ry=175.773637, rz=18.533291, fatherId=world[0]}
  [353] = {x=-3.1E-05, y=-51.810819, z=-2E-06, rx=0.30082, ry=175.773637, rz=18.533295, fatherId=world[0]}
  [354] = {x=-3.1E-05, y=-51.957592, z=-2E-06, rx=0.300816, ry=175.773636, rz=18.533298, fatherId=world[0]}
  [355] = {x=-3.1E-05, y=-52.104365, z=-2E-06, rx=0.300813, ry=175.773636, rz=18.533301, fatherId=world[0]}
  [356] = {x=-3.1E-05, y=-52.251138, z=-2E-06, rx=0.30081, ry=175.773636, rz=18.533304, fatherId=world[0]}
  [357] = {x=-3.1E-05, y=-52.39791, z=-2E-06, rx=0.300807, ry=175.773636, rz=18.533307, fatherId=world[0]}
  [358] = {x=-3.1E-05, y=-52.544683, z=-2E-06, rx=0.300803, ry=175.773636, rz=18.533311, fatherId=world[0]}
  [359] = {x=-3.1E-05, y=-52.691456, z=-2E-06, rx=0.3008, ry=175.773636, rz=18.533314, fatherId=world[0]}
  [360] = {x=-3.2E-05, y=-52.838229, z=-2E-06, rx=0.300797, ry=175.773636, rz=18.533317, fatherId=world[0]}
  [361] = {x=-3.2E-05, y=-52.985002, z=-2E-06, rx=0.300794, ry=175.773636, rz=18.53332, fatherId=world[0]}
  [362] = {x=-3.2E-05, y=-53.131775, z=-2E-06, rx=0.30079, ry=175.773636, rz=18.533324, fatherId=world[0]}
  [363] = {x=-3.2E-05, y=-53.278548, z=-2E-06, rx=0.300787, ry=175.773636, rz=18.533327, fatherId=world[0]}
  [364] = {x=-3.2E-05, y=-53.42532, z=-2E-06, rx=0.300784, ry=175.773635, rz=18.53333, fatherId=world[0]}
  [365] = {x=-3.2E-05, y=-53.572093, z=-2E-06, rx=0.300781, ry=175.773635, rz=18.533333, fatherId=world[0]}
  [366] = {x=-3.2E-05, y=-53.718866, z=-2E-06, rx=0.300778, ry=175.773635, rz=18.533336, fatherId=world[0]}
  [367] = {x=-3.2E-05, y=-53.865639, z=-3E-06, rx=0.300774, ry=175.773635, rz=18.53334, fatherId=world[0]}
  [368] = {x=-3.2E-05, y=-53.865639, z=-3E-06, rx=0.300774, ry=175.773635, rz=18.53334, fatherId=world[0]}
  [369] = {x=-3.2E-05, y=-54.012536, z=-3E-06, rx=0.30077, ry=175.773635, rz=18.533343, fatherId=world[0]}
  [370] = {x=-3.2E-05, y=-54.159433, z=-3E-06, rx=0.300767, ry=175.773635, rz=18.533347, fatherId=world[0]}
  [371] = {x=-3.3E-05, y=-54.30633, z=-3E-06, rx=0.300763, ry=175.773635, rz=18.533351, fatherId=world[0]}
  [372] = {x=-3.3E-05, y=-54.453228, z=-3E-06, rx=0.300759, ry=175.773635, rz=18.533355, fatherId=world[0]}
  [373] = {x=-3.3E-05, y=-54.600125, z=-3E-06, rx=0.300755, ry=175.773635, rz=18.533359, fatherId=world[0]}
  [374] = {x=-3.3E-05, y=-54.747022, z=-3E-06, rx=0.300751, ry=175.773635, rz=18.533362, fatherId=world[0]}
  [375] = {x=-3.3E-05, y=-54.893919, z=-3E-06, rx=0.300748, ry=175.773635, rz=18.533366, fatherId=world[0]}
  [376] = {x=-3.3E-05, y=-55.040816, z=-3E-06, rx=0.300744, ry=175.773635, rz=18.53337, fatherId=world[0]}
  [377] = {x=-3.3E-05, y=-55.187713, z=-3E-06, rx=0.30074, ry=175.773635, rz=18.533374, fatherId=world[0]}
  [378] = {x=-3.3E-05, y=-55.33461, z=-3E-06, rx=0.300736, ry=175.773635, rz=18.533378, fatherId=world[0]}
  [379] = {x=-3.3E-05, y=-55.481508, z=-3E-06, rx=0.300733, ry=175.773634, rz=18.533381, fatherId=world[0]}
  [380] = {x=-3.3E-05, y=-55.628405, z=-3E-06, rx=0.300729, ry=175.773634, rz=18.533385, fatherId=world[0]}
  [381] = {x=-3.3E-05, y=-55.775302, z=-3E-06, rx=0.300725, ry=175.773634, rz=18.533389, fatherId=world[0]}
  [382] = {x=-3.3E-05, y=-55.922199, z=-3E-06, rx=0.300721, ry=175.773634, rz=18.533393, fatherId=world[0]}
  [383] = {x=-3.3E-05, y=-56.069096, z=-3E-06, rx=0.300718, ry=175.773634, rz=18.533396, fatherId=world[0]}
  [384] = {x=-3.3E-05, y=-56.215993, z=-3E-06, rx=0.300714, ry=175.773634, rz=18.5334, fatherId=world[0]}
  [385] = {x=-3.3E-05, y=-56.36289, z=-3E-06, rx=0.30071, ry=175.773634, rz=18.533404, fatherId=world[0]}
  [386] = {x=-3.3E-05, y=-56.509788, z=-3E-06, rx=0.300706, ry=175.773634, rz=18.533407, fatherId=world[0]}
  [387] = {x=-3.3E-05, y=-56.656685, z=-3E-06, rx=0.300703, ry=175.773634, rz=18.533411, fatherId=world[0]}
  [388] = {x=-3.3E-05, y=-56.803582, z=-3E-06, rx=0.300699, ry=175.773634, rz=18.533415, fatherId=world[0]}
  [389] = {x=-3.4E-05, y=-56.950479, z=-3E-06, rx=0.300695, ry=175.773634, rz=18.533419, fatherId=world[0]}
  [390] = {x=-3.4E-05, y=-57.097376, z=-3E-06, rx=0.300692, ry=175.773634, rz=18.533422, fatherId=world[0]}
  [391] = {x=-3.4E-05, y=-57.244273, z=-3E-06, rx=0.300688, ry=175.773634, rz=18.533426, fatherId=world[0]}
  [392] = {x=-3.4E-05, y=-57.39117, z=-3E-06, rx=0.300684, ry=175.773634, rz=18.53343, fatherId=world[0]}
  [393] = {x=-3.4E-05, y=-57.538068, z=-3E-06, rx=0.30068, ry=175.773634, rz=18.533433, fatherId=world[0]}
  [394] = {x=-3.4E-05, y=-57.684965, z=-3E-06, rx=0.300677, ry=175.773634, rz=18.533437, fatherId=world[0]}
  [395] = {x=-3.4E-05, y=-57.831862, z=-3E-06, rx=0.300673, ry=175.773633, rz=18.533441, fatherId=world[0]}
  [396] = {x=-3.4E-05, y=-57.978759, z=-3E-06, rx=0.300669, ry=175.773633, rz=18.533445, fatherId=world[0]}
  [397] = {x=-3.4E-05, y=-58.125656, z=-3E-06, rx=0.300666, ry=175.773633, rz=18.533448, fatherId=world[0]}
  [398] = {x=-3.4E-05, y=-58.272553, z=-3E-06, rx=0.300662, ry=175.773633, rz=18.533452, fatherId=world[0]}
  [399] = {x=-3.4E-05, y=-58.419451, z=-3E-06, rx=0.300658, ry=175.773633, rz=18.533456, fatherId=world[0]}
  [400] = {x=-3.4E-05, y=-58.566348, z=-3E-06, rx=0.300655, ry=175.773633, rz=18.533459, fatherId=world[0]}
  [401] = {x=-3.4E-05, y=-58.713245, z=-3E-06, rx=0.300651, ry=175.773633, rz=18.533463, fatherId=world[0]}
  [402] = {x=-3.4E-05, y=-58.860142, z=-3E-06, rx=0.300647, ry=175.773633, rz=18.533467, fatherId=world[0]}
  [403] = {x=-3.4E-05, y=-59.007039, z=-3E-06, rx=0.300644, ry=175.773633, rz=18.53347, fatherId=world[0]}
  [404] = {x=-3.4E-05, y=-59.153936, z=-3E-06, rx=0.30064, ry=175.773633, rz=18.533474, fatherId=world[0]}
  [405] = {x=-3.4E-05, y=-59.300833, z=-3E-06, rx=0.300636, ry=175.773633, rz=18.533477, fatherId=world[0]}
  [406] = {x=-3.4E-05, y=-59.447731, z=-3E-06, rx=0.300633, ry=175.773633, rz=18.533481, fatherId=world[0]}
  [407] = {x=-3.5E-05, y=-59.594628, z=-3E-06, rx=0.300629, ry=175.773633, rz=18.533485, fatherId=world[0]}
  [408] = {x=-3.5E-05, y=-59.741525, z=-3E-06, rx=0.300626, ry=175.773633, rz=18.533488, fatherId=world[0]}
  [409] = {x=-3.5E-05, y=-59.888422, z=-3E-06, rx=0.300622, ry=175.773633, rz=18.533492, fatherId=world[0]}
  [410] = {x=-3.5E-05, y=-60.035319, z=-3E-06, rx=0.300618, ry=175.773633, rz=18.533496, fatherId=world[0]}
  [411] = {x=-3.5E-05, y=-60.182216, z=-3E-06, rx=0.300615, ry=175.773633, rz=18.533499, fatherId=world[0]}
  [412] = {x=-3.5E-05, y=-60.329113, z=-3E-06, rx=0.300611, ry=175.773633, rz=18.533503, fatherId=world[0]}
  [413] = {x=-3.5E-05, y=-60.476011, z=-3E-06, rx=0.300607, ry=175.773633, rz=18.533506, fatherId=world[0]}
  [414] = {x=-3.5E-05, y=-60.622908, z=-3E-06, rx=0.300604, ry=175.773633, rz=18.53351, fatherId=world[0]}
  [415] = {x=-3.5E-05, y=-60.769805, z=-3E-06, rx=0.3006, ry=175.773632, rz=18.533514, fatherId=world[0]}
  [416] = {x=-3.5E-05, y=-60.916702, z=-3E-06, rx=0.300597, ry=175.773632, rz=18.533517, fatherId=world[0]}
  [417] = {x=-3.5E-05, y=-61.063599, z=-3E-06, rx=0.300593, ry=175.773632, rz=18.533521, fatherId=world[0]}
  [418] = {x=-3.5E-05, y=-61.210496, z=-3E-06, rx=0.30059, ry=175.773632, rz=18.533524, fatherId=world[0]}
  [419] = {x=-3.5E-05, y=-61.357393, z=-3E-06, rx=0.300586, ry=175.773632, rz=18.533528, fatherId=world[0]}
  [420] = {x=-3.5E-05, y=-61.504291, z=-3E-06, rx=0.300582, ry=175.773632, rz=18.533532, fatherId=world[0]}
  [421] = {x=-3.5E-05, y=-61.651188, z=-3E-06, rx=0.300579, ry=175.773632, rz=18.533535, fatherId=world[0]}
  [422] = {x=-3.5E-05, y=-61.798085, z=-3E-06, rx=0.300575, ry=175.773632, rz=18.533539, fatherId=world[0]}
  [423] = {x=-3.5E-05, y=-61.944982, z=-3E-06, rx=0.300572, ry=175.773632, rz=18.533542, fatherId=world[0]}
  [424] = {x=-3.5E-05, y=-62.091879, z=-3E-06, rx=0.300568, ry=175.773632, rz=18.533546, fatherId=world[0]}
  [425] = {x=-3.5E-05, y=-62.238776, z=-3E-06, rx=0.300565, ry=175.773632, rz=18.533549, fatherId=world[0]}
  [426] = {x=-3.6E-05, y=-62.385673, z=-3E-06, rx=0.300561, ry=175.773632, rz=18.533553, fatherId=world[0]}
  [427] = {x=-3.6E-05, y=-62.532571, z=-3E-06, rx=0.300557, ry=175.773632, rz=18.533556, fatherId=world[0]}
  [428] = {x=-3.6E-05, y=-62.679468, z=-3E-06, rx=0.300554, ry=175.773632, rz=18.53356, fatherId=world[0]}
  [429] = {x=-3.6E-05, y=-62.826365, z=-3E-06, rx=0.30055, ry=175.773632, rz=18.533564, fatherId=world[0]}
  [430] = {x=-3.6E-05, y=-62.973262, z=-3E-06, rx=0.300547, ry=175.773632, rz=18.533567, fatherId=world[0]}
  [431] = {x=-3.6E-05, y=-63.120159, z=-3E-06, rx=0.300543, ry=175.773632, rz=18.533571, fatherId=world[0]}
  [432] = {x=-3.6E-05, y=-63.267056, z=-3E-06, rx=0.30054, ry=175.773632, rz=18.533574, fatherId=world[0]}
  [433] = {x=-3.6E-05, y=-63.413953, z=-3E-06, rx=0.300536, ry=175.773632, rz=18.533578, fatherId=world[0]}
  [434] = {x=-3.6E-05, y=-63.560851, z=-3E-06, rx=0.300533, ry=175.773632, rz=18.533581, fatherId=world[0]}
  [435] = {x=-3.6E-05, y=-63.707748, z=-3E-06, rx=0.300529, ry=175.773632, rz=18.533585, fatherId=world[0]}
  [436] = {x=-3.6E-05, y=-63.854645, z=-3E-06, rx=0.300526, ry=175.773632, rz=18.533588, fatherId=world[0]}
  [437] = {x=-3.6E-05, y=-64.001542, z=-3E-06, rx=0.300522, ry=175.773631, rz=18.533592, fatherId=world[0]}
  [438] = {x=-3.6E-05, y=-64.148439, z=-3E-06, rx=0.300519, ry=175.773631, rz=18.533595, fatherId=world[0]}
  [439] = {x=-3.6E-05, y=-64.295336, z=-3E-06, rx=0.300515, ry=175.773631, rz=18.533599, fatherId=world[0]}
  [440] = {x=-3.6E-05, y=-64.442233, z=-3E-06, rx=0.300512, ry=175.773631, rz=18.533602, fatherId=world[0]}
  [441] = {x=-3.6E-05, y=-64.589131, z=-3E-06, rx=0.300508, ry=175.773631, rz=18.533606, fatherId=world[0]}
  [442] = {x=-3.6E-05, y=-64.736028, z=-3E-06, rx=0.300505, ry=175.773631, rz=18.533609, fatherId=world[0]}
  [443] = {x=-3.6E-05, y=-64.882925, z=-3E-06, rx=0.300501, ry=175.773631, rz=18.533613, fatherId=world[0]}
  [444] = {x=-3.6E-05, y=-65.029822, z=-3E-06, rx=0.300498, ry=175.773631, rz=18.533616, fatherId=world[0]}
  [445] = {x=-3.7E-05, y=-65.176719, z=-3E-06, rx=0.300495, ry=175.773631, rz=18.533619, fatherId=world[0]}
  [446] = {x=-3.7E-05, y=-65.323616, z=-3E-06, rx=0.300491, ry=175.773631, rz=18.533623, fatherId=world[0]}
  [447] = {x=-3.7E-05, y=-65.470514, z=-3E-06, rx=0.300488, ry=175.773631, rz=18.533626, fatherId=world[0]}
  [448] = {x=-3.7E-05, y=-65.617411, z=-3E-06, rx=0.300484, ry=175.773631, rz=18.53363, fatherId=world[0]}
  [449] = {x=-3.7E-05, y=-65.764308, z=-3E-06, rx=0.300481, ry=175.773631, rz=18.533633, fatherId=world[0]}
  [450] = {x=-3.7E-05, y=-65.911205, z=-3E-06, rx=0.300477, ry=175.773631, rz=18.533637, fatherId=world[0]}
  [451] = {x=-3.7E-05, y=-66.058102, z=-3E-06, rx=0.300474, ry=175.773631, rz=18.53364, fatherId=world[0]}
  [452] = {x=-3.7E-05, y=-66.204999, z=-3E-06, rx=0.30047, ry=175.773631, rz=18.533644, fatherId=world[0]}
  [453] = {x=-3.7E-05, y=-66.351896, z=-3E-06, rx=0.300467, ry=175.773631, rz=18.533647, fatherId=world[0]}
  [454] = {x=-3.7E-05, y=-66.498794, z=-3E-06, rx=0.300464, ry=175.773631, rz=18.53365, fatherId=world[0]}
  [455] = {x=-3.7E-05, y=-66.645691, z=-3E-06, rx=0.30046, ry=175.773631, rz=18.533654, fatherId=world[0]}
  [456] = {x=-3.7E-05, y=-66.792588, z=-3E-06, rx=0.300457, ry=175.773631, rz=18.533657, fatherId=world[0]}
  [457] = {x=-3.7E-05, y=-66.939485, z=-3E-06, rx=0.300453, ry=175.773631, rz=18.533661, fatherId=world[0]}
  [458] = {x=-3.7E-05, y=-67.086382, z=-3E-06, rx=0.30045, ry=175.773631, rz=18.533664, fatherId=world[0]}
  [459] = {x=-3.7E-05, y=-67.233279, z=-3E-06, rx=0.300447, ry=175.773631, rz=18.533668, fatherId=world[0]}
  [460] = {x=-3.7E-05, y=-67.380176, z=-3E-06, rx=0.300443, ry=175.773631, rz=18.533671, fatherId=world[0]}
  [461] = {x=-3.7E-05, y=-67.527074, z=-3E-06, rx=0.30044, ry=175.773631, rz=18.533674, fatherId=world[0]}
  [462] = {x=-3.7E-05, y=-67.673971, z=-3E-06, rx=0.300436, ry=175.773631, rz=18.533678, fatherId=world[0]}
  [463] = {x=-3.7E-05, y=-67.820868, z=-3E-06, rx=0.300433, ry=175.773631, rz=18.533681, fatherId=world[0]}
  [464] = {x=-3.8E-05, y=-67.967765, z=-3E-06, rx=0.30043, ry=175.773631, rz=18.533684, fatherId=world[0]}
  [465] = {x=-3.8E-05, y=-68.114662, z=-3E-06, rx=0.300426, ry=175.773631, rz=18.533688, fatherId=world[0]}
  [466] = {x=-3.8E-05, y=-68.261559, z=-3E-06, rx=0.300423, ry=175.773631, rz=18.533691, fatherId=world[0]}
  [467] = {x=-3.8E-05, y=-68.408456, z=-3E-06, rx=0.30042, ry=175.77363, rz=18.533695, fatherId=world[0]}
  [468] = {x=-3.8E-05, y=-68.555354, z=-3E-06, rx=0.300416, ry=175.77363, rz=18.533698, fatherId=world[0]}
  [469] = {x=-3.8E-05, y=-68.702251, z=-3E-06, rx=0.300413, ry=175.77363, rz=18.533701, fatherId=world[0]}
  [470] = {x=-3.8E-05, y=-68.849148, z=-3E-06, rx=0.300409, ry=175.77363, rz=18.533705, fatherId=world[0]}
  [471] = {x=-3.8E-05, y=-68.996045, z=-3E-06, rx=0.300406, ry=175.77363, rz=18.533708, fatherId=world[0]}
  [472] = {x=-3.8E-05, y=-69.142942, z=-3E-06, rx=0.300403, ry=175.77363, rz=18.533711, fatherId=world[0]}
  [473] = {x=-3.8E-05, y=-69.289839, z=-3E-06, rx=0.300399, ry=175.77363, rz=18.533715, fatherId=world[0]}
  [474] = {x=-3.8E-05, y=-69.436736, z=-3E-06, rx=0.300396, ry=175.77363, rz=18.533718, fatherId=world[0]}
  [475] = {x=-3.8E-05, y=-69.583634, z=-3E-06, rx=0.300393, ry=175.77363, rz=18.533721, fatherId=world[0]}
  [476] = {x=-3.8E-05, y=-69.730531, z=-3E-06, rx=0.30039, ry=175.77363, rz=18.533725, fatherId=world[0]}
  [477] = {x=-3.8E-05, y=-69.877428, z=-3E-06, rx=0.300386, ry=175.77363, rz=18.533728, fatherId=world[0]}
  [478] = {x=-3.8E-05, y=-70.024325, z=-3E-06, rx=0.300383, ry=175.77363, rz=18.533731, fatherId=world[0]}
  [479] = {x=-3.8E-05, y=-70.171222, z=-3E-06, rx=0.30038, ry=175.77363, rz=18.533735, fatherId=world[0]}
  [480] = {x=-3.8E-05, y=-70.318119, z=-4E-06, rx=0.300376, ry=175.77363, rz=18.533738, fatherId=world[0]}
  [481] = {x=-3.8E-05, y=-70.465016, z=-4E-06, rx=0.300373, ry=175.77363, rz=18.533741, fatherId=world[0]}
  [482] = {x=-3.8E-05, y=-70.611914, z=-4E-06, rx=0.30037, ry=175.77363, rz=18.533744, fatherId=world[0]}
  [483] = {x=-3.8E-05, y=-70.758811, z=-4E-06, rx=0.300366, ry=175.77363, rz=18.533748, fatherId=world[0]}
  [484] = {x=-3.8E-05, y=-70.905708, z=-4E-06, rx=0.300363, ry=175.77363, rz=18.533751, fatherId=world[0]}
  [485] = {x=-3.9E-05, y=-71.052605, z=-4E-06, rx=0.30036, ry=175.77363, rz=18.533754, fatherId=world[0]}
  [486] = {x=-3.9E-05, y=-71.199502, z=-4E-06, rx=0.300357, ry=175.77363, rz=18.533758, fatherId=world[0]}
  [487] = {x=-3.9E-05, y=-71.346399, z=-4E-06, rx=0.300353, ry=175.77363, rz=18.533761, fatherId=world[0]}
  [488] = {x=-3.9E-05, y=-71.493296, z=-4E-06, rx=0.30035, ry=175.77363, rz=18.533764, fatherId=world[0]}
  [489] = {x=-3.9E-05, y=-71.640194, z=-4E-06, rx=0.300347, ry=175.77363, rz=18.533767, fatherId=world[0]}
  [490] = {x=-3.9E-05, y=-71.787091, z=-4E-06, rx=0.300344, ry=175.77363, rz=18.533771, fatherId=world[0]}
  [491] = {x=-3.9E-05, y=-71.933988, z=-4E-06, rx=0.30034, ry=175.77363, rz=18.533774, fatherId=world[0]}
  [492] = {x=-3.9E-05, y=-72.080885, z=-4E-06, rx=0.300337, ry=175.77363, rz=18.533777, fatherId=world[0]}
  [493] = {x=-3.9E-05, y=-72.227782, z=-4E-06, rx=0.300334, ry=175.77363, rz=18.53378, fatherId=world[0]}
  [494] = {x=-3.9E-05, y=-72.374679, z=-4E-06, rx=0.300331, ry=175.77363, rz=18.533784, fatherId=world[0]}
  [495] = {x=-3.9E-05, y=-72.521576, z=-4E-06, rx=0.300327, ry=175.77363, rz=18.533787, fatherId=world[0]}
  [496] = {x=-3.9E-05, y=-72.668474, z=-4E-06, rx=0.300324, ry=175.77363, rz=18.53379, fatherId=world[0]}
  [497] = {x=-3.9E-05, y=-72.815371, z=-4E-06, rx=0.300321, ry=175.77363, rz=18.533793, fatherId=world[0]}
  [498] = {x=-3.9E-05, y=-72.962268, z=-4E-06, rx=0.300318, ry=175.77363, rz=18.533797, fatherId=world[0]}
  [499] = {x=-3.9E-05, y=-73.109165, z=-4E-06, rx=0.300314, ry=175.77363, rz=18.5338, fatherId=world[0]}
  [500] = {x=-3.9E-05, y=-73.256062, z=-4E-06, rx=0.300311, ry=175.77363, rz=18.533803, fatherId=world[0]}
  [501] = {x=-3.9E-05, y=-73.402959, z=-4E-06, rx=0.300308, ry=175.77363, rz=18.533806, fatherId=world[0]}
  [502] = {x=-3.9E-05, y=-73.549857, z=-4E-06, rx=0.300305, ry=175.77363, rz=18.53381, fatherId=world[0]}
  [503] = {x=-3.9E-05, y=-73.696754, z=-4E-06, rx=0.300302, ry=175.77363, rz=18.533813, fatherId=world[0]}
  [504] = {x=-3.9E-05, y=-73.843651, z=-4E-06, rx=0.300298, ry=175.77363, rz=18.533816, fatherId=world[0]}
  [505] = {x=-3.9E-05, y=-73.990548, z=-4E-06, rx=0.300295, ry=175.77363, rz=18.533819, fatherId=world[0]}
  [506] = {x=-4E-05, y=-74.137445, z=-4E-06, rx=0.300292, ry=175.77363, rz=18.533822, fatherId=world[0]}
  [507] = {x=-4E-05, y=-74.284342, z=-4E-06, rx=0.300289, ry=175.77363, rz=18.533825, fatherId=world[0]}
  [508] = {x=-4E-05, y=-74.431239, z=-4E-06, rx=0.300286, ry=175.77363, rz=18.533829, fatherId=world[0]}
  [509] = {x=-4E-05, y=-74.578137, z=-4E-06, rx=0.300283, ry=175.77363, rz=18.533832, fatherId=world[0]}
  [510] = {x=-4E-05, y=-74.725034, z=-4E-06, rx=0.300279, ry=175.77363, rz=18.533835, fatherId=world[0]}
  [511] = {x=-4E-05, y=-74.871931, z=-4E-06, rx=0.300276, ry=175.77363, rz=18.533838, fatherId=world[0]}
  [512] = {x=-4E-05, y=-75.018828, z=-4E-06, rx=0.300273, ry=175.77363, rz=18.533841, fatherId=world[0]}
  [513] = {x=-4E-05, y=-75.165725, z=-4E-06, rx=0.30027, ry=175.77363, rz=18.533844, fatherId=world[0]}
  [514] = {x=-4E-05, y=-75.312622, z=-4E-06, rx=0.300267, ry=175.77363, rz=18.533848, fatherId=world[0]}
  [515] = {x=-4E-05, y=-75.459519, z=-4E-06, rx=0.300264, ry=175.77363, rz=18.533851, fatherId=world[0]}
  [516] = {x=-4E-05, y=-75.606417, z=-4E-06, rx=0.300261, ry=175.77363, rz=18.533854, fatherId=world[0]}
  [517] = {x=-4E-05, y=-75.753314, z=-4E-06, rx=0.300257, ry=175.77363, rz=18.533857, fatherId=world[0]}
  [518] = {x=-4E-05, y=-75.900211, z=-4E-06, rx=0.300254, ry=175.77363, rz=18.53386, fatherId=world[0]}
  [519] = {x=-4E-05, y=-76.047108, z=-4E-06, rx=0.300251, ry=175.77363, rz=18.533863, fatherId=world[0]}
  [520] = {x=-4E-05, y=-76.194005, z=-4E-06, rx=0.300248, ry=175.77363, rz=18.533866, fatherId=world[0]}
  [521] = {x=-4E-05, y=-76.340902, z=-4E-06, rx=0.300245, ry=175.77363, rz=18.53387, fatherId=world[0]}
  [522] = {x=-4E-05, y=-76.487799, z=-4E-06, rx=0.300242, ry=175.77363, rz=18.533873, fatherId=world[0]}
  [523] = {x=-4E-05, y=-76.634697, z=-4E-06, rx=0.300239, ry=175.77363, rz=18.533876, fatherId=world[0]}
  [524] = {x=-4E-05, y=-76.781594, z=-4E-06, rx=0.300236, ry=175.77363, rz=18.533879, fatherId=world[0]}
  [525] = {x=-4E-05, y=-76.928491, z=-4E-06, rx=0.300232, ry=175.77363, rz=18.533882, fatherId=world[0]}
  [526] = {x=-4E-05, y=-77.075388, z=-4E-06, rx=0.300229, ry=175.77363, rz=18.533885, fatherId=world[0]}
  [527] = {x=-4.1E-05, y=-77.222285, z=-4E-06, rx=0.300226, ry=175.77363, rz=18.533888, fatherId=world[0]}
  [528] = {x=-4.1E-05, y=-77.369182, z=-4E-06, rx=0.300223, ry=175.77363, rz=18.533891, fatherId=world[0]}
  [529] = {x=-4.1E-05, y=-77.516079, z=-4E-06, rx=0.30022, ry=175.77363, rz=18.533894, fatherId=world[0]}
  [530] = {x=-4.1E-05, y=-77.662977, z=-4E-06, rx=0.300217, ry=175.77363, rz=18.533898, fatherId=world[0]}
  [531] = {x=-4.1E-05, y=-77.809874, z=-4E-06, rx=0.300214, ry=175.77363, rz=18.533901, fatherId=world[0]}
  [532] = {x=-4.1E-05, y=-77.956771, z=-4E-06, rx=0.300211, ry=175.77363, rz=18.533904, fatherId=world[0]}
  [533] = {x=-4.1E-05, y=-78.103668, z=-4E-06, rx=0.300208, ry=175.77363, rz=18.533907, fatherId=world[0]}
  [534] = {x=-4.1E-05, y=-78.250565, z=-4E-06, rx=0.300205, ry=175.77363, rz=18.53391, fatherId=world[0]}
  [535] = {x=-4.1E-05, y=-78.397462, z=-4E-06, rx=0.300202, ry=175.77363, rz=18.533913, fatherId=world[0]}
  [536] = {x=-4.1E-05, y=-78.544359, z=-4E-06, rx=0.300199, ry=175.77363, rz=18.533916, fatherId=world[0]}
  [537] = {x=-4.1E-05, y=-78.691257, z=-4E-06, rx=0.300196, ry=175.77363, rz=18.533919, fatherId=world[0]}
  [538] = {x=-4.1E-05, y=-78.838154, z=-4E-06, rx=0.300193, ry=175.77363, rz=18.533922, fatherId=world[0]}
  [539] = {x=-4.1E-05, y=-78.985051, z=-4E-06, rx=0.30019, ry=175.77363, rz=18.533925, fatherId=world[0]}
  [540] = {x=-4.1E-05, y=-79.131948, z=-4E-06, rx=0.300187, ry=175.77363, rz=18.533928, fatherId=world[0]}
  [541] = {x=-4.1E-05, y=-79.278845, z=-4E-06, rx=0.300184, ry=175.77363, rz=18.533931, fatherId=world[0]}
  [542] = {x=-4.1E-05, y=-79.425742, z=-4E-06, rx=0.300181, ry=175.77363, rz=18.533934, fatherId=world[0]}
  [543] = {x=-4.1E-05, y=-79.572639, z=-4E-06, rx=0.300178, ry=175.77363, rz=18.533937, fatherId=world[0]}
  [544] = {x=-4.1E-05, y=-79.719537, z=-4E-06, rx=0.300175, ry=175.77363, rz=18.53394, fatherId=world[0]}
  [545] = {x=-4.1E-05, y=-79.866434, z=-4E-06, rx=0.300172, ry=175.77363, rz=18.533943, fatherId=world[0]}
  [546] = {x=-4.1E-05, y=-80.013331, z=-4E-06, rx=0.300169, ry=175.77363, rz=18.533946, fatherId=world[0]}
  [547] = {x=-4.1E-05, y=-80.160228, z=-4E-06, rx=0.300166, ry=175.77363, rz=18.533949, fatherId=world[0]}
  [548] = {x=-4.1E-05, y=-80.307125, z=-4E-06, rx=0.300163, ry=175.77363, rz=18.533952, fatherId=world[0]}
  [549] = {x=-4.2E-05, y=-80.454022, z=-4E-06, rx=0.30016, ry=175.77363, rz=18.533955, fatherId=world[0]}
  [550] = {x=-4.2E-05, y=-80.60092, z=-4E-06, rx=0.300157, ry=175.77363, rz=18.533958, fatherId=world[0]}
  [551] = {x=-4.2E-05, y=-80.747817, z=-4E-06, rx=0.300154, ry=175.77363, rz=18.533961, fatherId=world[0]}
  [552] = {x=-4.2E-05, y=-80.894714, z=-4E-06, rx=0.300151, ry=175.77363, rz=18.533964, fatherId=world[0]}
  [553] = {x=-4.2E-05, y=-81.041611, z=-4E-06, rx=0.300148, ry=175.77363, rz=18.533967, fatherId=world[0]}
  [554] = {x=-4.2E-05, y=-81.188508, z=-4E-06, rx=0.300145, ry=175.77363, rz=18.53397, fatherId=world[0]}
  [555] = {x=-4.2E-05, y=-81.335405, z=-4E-06, rx=0.300142, ry=175.77363, rz=18.533973, fatherId=world[0]}
  [556] = {x=-4.2E-05, y=-81.482302, z=-4E-06, rx=0.300139, ry=175.77363, rz=18.533976, fatherId=world[0]}
  [557] = {x=-4.2E-05, y=-81.6292, z=-4E-06, rx=0.300136, ry=175.77363, rz=18.533979, fatherId=world[0]}
  [558] = {x=-4.2E-05, y=-81.776097, z=-4E-06, rx=0.300133, ry=175.77363, rz=18.533982, fatherId=world[0]}
  [559] = {x=-4.2E-05, y=-81.922994, z=-4E-06, rx=0.30013, ry=175.77363, rz=18.533985, fatherId=world[0]}
  [560] = {x=-4.2E-05, y=-82.069891, z=-4E-06, rx=0.300127, ry=175.77363, rz=18.533988, fatherId=world[0]}
  [561] = {x=-4.2E-05, y=-82.216788, z=-4E-06, rx=0.300124, ry=175.77363, rz=18.533991, fatherId=world[0]}
  [562] = {x=-4.2E-05, y=-82.363685, z=-4E-06, rx=0.300121, ry=175.77363, rz=18.533994, fatherId=world[0]}
  [563] = {x=-4.2E-05, y=-82.510582, z=-4E-06, rx=0.300118, ry=175.77363, rz=18.533997, fatherId=world[0]}
  [564] = {x=-4.2E-05, y=-82.65748, z=-4E-06, rx=0.300115, ry=175.77363, rz=18.534, fatherId=world[0]}
  [565] = {x=-4.2E-05, y=-82.804377, z=-4E-06, rx=0.300112, ry=175.77363, rz=18.534003, fatherId=world[0]}
  [566] = {x=-4.2E-05, y=-82.951274, z=-4E-06, rx=0.30011, ry=175.77363, rz=18.534005, fatherId=world[0]}
  [567] = {x=-4.2E-05, y=-83.098171, z=-4E-06, rx=0.300107, ry=175.77363, rz=18.534008, fatherId=world[0]}
  [568] = {x=-4.2E-05, y=-83.245068, z=-4E-06, rx=0.300104, ry=175.77363, rz=18.534011, fatherId=world[0]}
  [569] = {x=-4.2E-05, y=-83.391965, z=-4E-06, rx=0.300101, ry=175.77363, rz=18.534014, fatherId=world[0]}
  [570] = {x=-4.2E-05, y=-83.538862, z=-4E-06, rx=0.300098, ry=175.77363, rz=18.534017, fatherId=world[0]}
  [571] = {x=-4.2E-05, y=-83.68576, z=-4E-06, rx=0.300095, ry=175.77363, rz=18.53402, fatherId=world[0]}
  [572] = {x=-4.2E-05, y=-83.832657, z=-4E-06, rx=0.300092, ry=175.77363, rz=18.534023, fatherId=world[0]}
  [573] = {x=-4.3E-05, y=-83.979554, z=-4E-06, rx=0.300089, ry=175.77363, rz=18.534026, fatherId=world[0]}
  [574] = {x=-4.3E-05, y=-84.126451, z=-4E-06, rx=0.300086, ry=175.77363, rz=18.534029, fatherId=world[0]}
  [575] = {x=-4.3E-05, y=-84.273348, z=-4E-06, rx=0.300084, ry=175.77363, rz=18.534032, fatherId=world[0]}
  [576] = {x=-4.3E-05, y=-84.420245, z=-4E-06, rx=0.300081, ry=175.77363, rz=18.534034, fatherId=world[0]}
  [577] = {x=-4.3E-05, y=-84.567142, z=-4E-06, rx=0.300078, ry=175.77363, rz=18.534037, fatherId=world[0]}
  [578] = {x=-4.3E-05, y=-84.71404, z=-4E-06, rx=0.300075, ry=175.77363, rz=18.53404, fatherId=world[0]}
  [579] = {x=-4.3E-05, y=-84.860937, z=-4E-06, rx=0.300072, ry=175.77363, rz=18.534043, fatherId=world[0]}
  [580] = {x=-4.3E-05, y=-85.007834, z=-4E-06, rx=0.300069, ry=175.77363, rz=18.534046, fatherId=world[0]}
  [581] = {x=-4.3E-05, y=-85.154731, z=-4E-06, rx=0.300066, ry=175.77363, rz=18.534049, fatherId=world[0]}
  [582] = {x=-4.3E-05, y=-85.301628, z=-5E-06, rx=0.300064, ry=175.77363, rz=18.534052, fatherId=world[0]}
  [583] = {x=-4.3E-05, y=-85.448525, z=-5E-06, rx=0.300061, ry=175.77363, rz=18.534054, fatherId=world[0]}
  [584] = {x=-4.3E-05, y=-85.595422, z=-5E-06, rx=0.300058, ry=175.77363, rz=18.534057, fatherId=world[0]}
  [585] = {x=-4.3E-05, y=-85.74232, z=-5E-06, rx=0.300055, ry=175.77363, rz=18.53406, fatherId=world[0]}
  [586] = {x=-4.3E-05, y=-85.889217, z=-5E-06, rx=0.300052, ry=175.77363, rz=18.534063, fatherId=world[0]}
  [587] = {x=-4.3E-05, y=-86.036114, z=-5E-06, rx=0.30005, ry=175.77363, rz=18.534066, fatherId=world[0]}
  [588] = {x=-4.3E-05, y=-86.183011, z=-5E-06, rx=0.300047, ry=175.77363, rz=18.534069, fatherId=world[0]}
  [589] = {x=-4.3E-05, y=-86.329908, z=-5E-06, rx=0.300044, ry=175.77363, rz=18.534071, fatherId=world[0]}
  [590] = {x=-4.3E-05, y=-86.476805, z=-5E-06, rx=0.300041, ry=175.77363, rz=18.534074, fatherId=world[0]}
  [591] = {x=-4.3E-05, y=-86.623702, z=-5E-06, rx=0.300038, ry=175.77363, rz=18.534077, fatherId=world[0]}
  [592] = {x=-4.3E-05, y=-86.7706, z=-5E-06, rx=0.300036, ry=175.77363, rz=18.53408, fatherId=world[0]}
  [593] = {x=-4.3E-05, y=-86.917497, z=-5E-06, rx=0.300033, ry=175.77363, rz=18.534083, fatherId=world[0]}
  [594] = {x=-4.3E-05, y=-87.064394, z=-5E-06, rx=0.30003, ry=175.77363, rz=18.534085, fatherId=world[0]}
  [595] = {x=-4.3E-05, y=-87.211291, z=-5E-06, rx=0.300027, ry=175.77363, rz=18.534088, fatherId=world[0]}
  [596] = {x=-4.3E-05, y=-87.358188, z=-5E-06, rx=0.300024, ry=175.77363, rz=18.534091, fatherId=world[0]}
  [597] = {x=-4.4E-05, y=-87.505085, z=-5E-06, rx=0.300022, ry=175.77363, rz=18.534094, fatherId=world[0]}
  [598] = {x=-4.4E-05, y=-87.651983, z=-5E-06, rx=0.300019, ry=175.77363, rz=18.534097, fatherId=world[0]}
  [599] = {x=-4.4E-05, y=-87.79888, z=-5E-06, rx=0.300016, ry=175.77363, rz=18.534099, fatherId=world[0]}
  [600] = {x=-4.4E-05, y=-87.945777, z=-5E-06, rx=0.300013, ry=175.77363, rz=18.534102, fatherId=world[0]}
  [601] = {x=-4.4E-05, y=-88.092674, z=-5E-06, rx=0.300011, ry=175.77363, rz=18.534105, fatherId=world[0]}
  [602] = {x=-4.4E-05, y=-88.239571, z=-5E-06, rx=0.300008, ry=175.77363, rz=18.534108, fatherId=world[0]}
  [603] = {x=-4.4E-05, y=-88.386468, z=-5E-06, rx=0.300005, ry=175.77363, rz=18.53411, fatherId=world[0]}
  [604] = {x=-4.4E-05, y=-88.533365, z=-5E-06, rx=0.300002, ry=175.77363, rz=18.534113, fatherId=world[0]}
  [605] = {x=-4.4E-05, y=-88.680263, z=-5E-06, rx=0.3, ry=175.77363, rz=18.534116, fatherId=world[0]}
  [606] = {x=-4.4E-05, y=-88.82716, z=-5E-06, rx=0.299997, ry=175.773631, rz=18.534119, fatherId=world[0]}
  [607] = {x=-4.4E-05, y=-88.974057, z=-5E-06, rx=0.299994, ry=175.773631, rz=18.534121, fatherId=world[0]}
  [608] = {x=-4.4E-05, y=-89.120954, z=-5E-06, rx=0.299992, ry=175.773631, rz=18.534124, fatherId=world[0]}
  [609] = {x=-4.4E-05, y=-89.267851, z=-5E-06, rx=0.299989, ry=175.773631, rz=18.534127, fatherId=world[0]}
  [610] = {x=-4.4E-05, y=-89.414748, z=-5E-06, rx=0.299986, ry=175.773631, rz=18.53413, fatherId=world[0]}
  [611] = {x=-4.4E-05, y=-89.561645, z=-5E-06, rx=0.299983, ry=175.773631, rz=18.534132, fatherId=world[0]}
  [612] = {x=-4.4E-05, y=-89.708543, z=-5E-06, rx=0.299981, ry=175.773631, rz=18.534135, fatherId=world[0]}
  [613] = {x=-4.4E-05, y=-89.85544, z=-5E-06, rx=0.299978, ry=175.773631, rz=18.534138, fatherId=world[0]}
  [614] = {x=-4.4E-05, y=-90.002337, z=-5E-06, rx=0.299975, ry=175.773631, rz=18.53414, fatherId=world[0]}
  [615] = {x=-4.4E-05, y=-90.149234, z=-5E-06, rx=0.299973, ry=175.773631, rz=18.534143, fatherId=world[0]}
  [616] = {x=-4.4E-05, y=-90.296131, z=-5E-06, rx=0.29997, ry=175.773631, rz=18.534146, fatherId=world[0]}
  [617] = {x=-4.4E-05, y=-90.443028, z=-5E-06, rx=0.299967, ry=175.773631, rz=18.534148, fatherId=world[0]}
  [618] = {x=-4.4E-05, y=-90.589925, z=-5E-06, rx=0.299965, ry=175.773631, rz=18.534151, fatherId=world[0]}
  [619] = {x=-4.4E-05, y=-90.736823, z=-5E-06, rx=0.299962, ry=175.773631, rz=18.534154, fatherId=world[0]}
  [620] = {x=-4.4E-05, y=-90.88372, z=-5E-06, rx=0.299959, ry=175.773631, rz=18.534157, fatherId=world[0]}
  [621] = {x=-4.4E-05, y=-91.030617, z=-5E-06, rx=0.299957, ry=175.773631, rz=18.534159, fatherId=world[0]}
  [622] = {x=-4.5E-05, y=-91.177514, z=-5E-06, rx=0.299954, ry=175.773631, rz=18.534162, fatherId=world[0]}
  [623] = {x=-4.5E-05, y=-91.324411, z=-5E-06, rx=0.299951, ry=175.773631, rz=18.534165, fatherId=world[0]}
  [624] = {x=-4.5E-05, y=-91.471308, z=-5E-06, rx=0.299949, ry=175.773631, rz=18.534167, fatherId=world[0]}
  [625] = {x=-4.5E-05, y=-91.618205, z=-5E-06, rx=0.299946, ry=175.773631, rz=18.53417, fatherId=world[0]}
  [626] = {x=-4.5E-05, y=-91.765103, z=-5E-06, rx=0.299943, ry=175.773631, rz=18.534173, fatherId=world[0]}
  [627] = {x=-4.5E-05, y=-91.912, z=-5E-06, rx=0.299941, ry=175.773631, rz=18.534175, fatherId=world[0]}
  [628] = {x=-4.5E-05, y=-92.058897, z=-5E-06, rx=0.299938, ry=175.773631, rz=18.534178, fatherId=world[0]}
  [629] = {x=-4.5E-05, y=-92.205794, z=-5E-06, rx=0.299936, ry=175.773631, rz=18.53418, fatherId=world[0]}
  [630] = {x=-4.5E-05, y=-92.352691, z=-5E-06, rx=0.299933, ry=175.773631, rz=18.534183, fatherId=world[0]}
  [631] = {x=-4.5E-05, y=-92.499588, z=-5E-06, rx=0.29993, ry=175.773631, rz=18.534186, fatherId=world[0]}
  [632] = {x=-4.5E-05, y=-92.646485, z=-5E-06, rx=0.299928, ry=175.773631, rz=18.534188, fatherId=world[0]}
  [633] = {x=-4.5E-05, y=-92.793383, z=-5E-06, rx=0.299925, ry=175.773631, rz=18.534191, fatherId=world[0]}
  [634] = {x=-4.5E-05, y=-92.94028, z=-5E-06, rx=0.299923, ry=175.773631, rz=18.534194, fatherId=world[0]}
  [635] = {x=-4.5E-05, y=-93.087177, z=-5E-06, rx=0.29992, ry=175.773631, rz=18.534196, fatherId=world[0]}
  [636] = {x=-4.5E-05, y=-93.234074, z=-5E-06, rx=0.299917, ry=175.773632, rz=18.534199, fatherId=world[0]}
  [637] = {x=-4.5E-05, y=-93.380971, z=-5E-06, rx=0.299915, ry=175.773632, rz=18.534201, fatherId=world[0]}
  [638] = {x=-4.5E-05, y=-93.527868, z=-5E-06, rx=0.299912, ry=175.773632, rz=18.534204, fatherId=world[0]}
  [639] = {x=-4.5E-05, y=-93.674765, z=-5E-06, rx=0.29991, ry=175.773632, rz=18.534207, fatherId=world[0]}
  [640] = {x=-4.5E-05, y=-93.821663, z=-5E-06, rx=0.299907, ry=175.773632, rz=18.534209, fatherId=world[0]}
  [641] = {x=-4.5E-05, y=-93.96856, z=-5E-06, rx=0.299904, ry=175.773632, rz=18.534212, fatherId=world[0]}
  [642] = {x=-4.5E-05, y=-94.115457, z=-5E-06, rx=0.299902, ry=175.773632, rz=18.534214, fatherId=world[0]}
  [643] = {x=-4.5E-05, y=-94.262354, z=-5E-06, rx=0.299899, ry=175.773632, rz=18.534217, fatherId=world[0]}
  [644] = {x=-4.5E-05, y=-94.409251, z=-5E-06, rx=0.299897, ry=175.773632, rz=18.534219, fatherId=world[0]}
  [645] = {x=-4.5E-05, y=-94.556148, z=-5E-06, rx=0.299894, ry=175.773632, rz=18.534222, fatherId=world[0]}
  [646] = {x=-4.5E-05, y=-94.703046, z=-5E-06, rx=0.299892, ry=175.773632, rz=18.534225, fatherId=world[0]}
  [647] = {x=-4.5E-05, y=-94.849943, z=-5E-06, rx=0.299889, ry=175.773632, rz=18.534227, fatherId=world[0]}
  [648] = {x=-4.5E-05, y=-94.99684, z=-5E-06, rx=0.299887, ry=175.773632, rz=18.53423, fatherId=world[0]}
  [649] = {x=-4.6E-05, y=-95.143737, z=-5E-06, rx=0.299884, ry=175.773632, rz=18.534232, fatherId=world[0]}
  [650] = {x=-4.6E-05, y=-95.290634, z=-5E-06, rx=0.299882, ry=175.773632, rz=18.534235, fatherId=world[0]}
  [651] = {x=-4.6E-05, y=-95.437531, z=-5E-06, rx=0.299879, ry=175.773632, rz=18.534237, fatherId=world[0]}
  [652] = {x=-4.6E-05, y=-95.584428, z=-5E-06, rx=0.299877, ry=175.773632, rz=18.53424, fatherId=world[0]}
  [653] = {x=-4.6E-05, y=-95.731326, z=-5E-06, rx=0.299874, ry=175.773632, rz=18.534242, fatherId=world[0]}
  [654] = {x=-4.6E-05, y=-95.878223, z=-5E-06, rx=0.299872, ry=175.773632, rz=18.534245, fatherId=world[0]}
  [655] = {x=-4.6E-05, y=-96.02512, z=-5E-06, rx=0.299869, ry=175.773632, rz=18.534247, fatherId=world[0]}
  [656] = {x=-4.6E-05, y=-96.172017, z=-5E-06, rx=0.299867, ry=175.773632, rz=18.53425, fatherId=world[0]}
  [657] = {x=-4.6E-05, y=-96.318914, z=-5E-06, rx=0.299864, ry=175.773632, rz=18.534252, fatherId=world[0]}
  [658] = {x=-4.6E-05, y=-96.465811, z=-5E-06, rx=0.299862, ry=175.773632, rz=18.534255, fatherId=world[0]}
  [659] = {x=-4.6E-05, y=-96.612708, z=-5E-06, rx=0.299859, ry=175.773633, rz=18.534258, fatherId=world[0]}
  [660] = {x=-4.6E-05, y=-96.759606, z=-5E-06, rx=0.299857, ry=175.773633, rz=18.53426, fatherId=world[0]}
  [661] = {x=-4.6E-05, y=-96.906503, z=-5E-06, rx=0.299854, ry=175.773633, rz=18.534262, fatherId=world[0]}
  [662] = {x=-4.6E-05, y=-97.0534, z=-5E-06, rx=0.299852, ry=175.773633, rz=18.534265, fatherId=world[0]}
  [663] = {x=-4.6E-05, y=-97.200297, z=-5E-06, rx=0.299849, ry=175.773633, rz=18.534267, fatherId=world[0]}
  [664] = {x=-4.6E-05, y=-97.347194, z=-5E-06, rx=0.299847, ry=175.773633, rz=18.53427, fatherId=world[0]}
  [665] = {x=-4.6E-05, y=-97.494091, z=-5E-06, rx=0.299844, ry=175.773633, rz=18.534272, fatherId=world[0]}
  [666] = {x=-4.6E-05, y=-97.640988, z=-5E-06, rx=0.299842, ry=175.773633, rz=18.534275, fatherId=world[0]}
  [667] = {x=-4.6E-05, y=-97.787886, z=-5E-06, rx=0.299839, ry=175.773633, rz=18.534277, fatherId=world[0]}
  [668] = {x=-4.6E-05, y=-97.934783, z=-5E-06, rx=0.299837, ry=175.773633, rz=18.53428, fatherId=world[0]}
  [669] = {x=-4.6E-05, y=-98.08168, z=-5E-06, rx=0.299834, ry=175.773633, rz=18.534282, fatherId=world[0]}
  [670] = {x=-4.6E-05, y=-98.228577, z=-5E-06, rx=0.299832, ry=175.773633, rz=18.534285, fatherId=world[0]}
  [671] = {x=-4.6E-05, y=-98.375474, z=-5E-06, rx=0.29983, ry=175.773633, rz=18.534287, fatherId=world[0]}
  [672] = {x=-4.6E-05, y=-98.522371, z=-5E-06, rx=0.299827, ry=175.773633, rz=18.53429, fatherId=world[0]}
  [673] = {x=-4.6E-05, y=-98.669268, z=-5E-06, rx=0.299825, ry=175.773633, rz=18.534292, fatherId=world[0]}
  [674] = {x=-4.6E-05, y=-98.816166, z=-5E-06, rx=0.299822, ry=175.773633, rz=18.534295, fatherId=world[0]}
  [675] = {x=-4.6E-05, y=-98.963063, z=-5E-06, rx=0.29982, ry=175.773633, rz=18.534297, fatherId=world[0]}
  [676] = {x=-4.6E-05, y=-99.10996, z=-6E-06, rx=0.299818, ry=175.773633, rz=18.534299, fatherId=world[0]}
  [677] = {x=-4.7E-05, y=-99.256857, z=-6E-06, rx=0.299815, ry=175.773633, rz=18.534302, fatherId=world[0]}
  [678] = {x=-4.7E-05, y=-99.403754, z=-6E-06, rx=0.299813, ry=175.773634, rz=18.534304, fatherId=world[0]}
  [679] = {x=-4.7E-05, y=-99.550651, z=-6E-06, rx=0.29981, ry=175.773634, rz=18.534307, fatherId=world[0]}
  [680] = {x=-4.7E-05, y=-99.697548, z=-6E-06, rx=0.299808, ry=175.773634, rz=18.534309, fatherId=world[0]}
  [681] = {x=-4.7E-05, y=-99.844446, z=-6E-06, rx=0.299806, ry=175.773634, rz=18.534311, fatherId=world[0]}
  [682] = {x=-4.7E-05, y=-99.991343, z=-6E-06, rx=0.299803, ry=175.773634, rz=18.534314, fatherId=world[0]}
  [683] = {x=-4.7E-05, y=-100.13824, z=-6E-06, rx=0.299801, ry=175.773634, rz=18.534316, fatherId=world[0]}
  [684] = {x=-4.7E-05, y=-100.285137, z=-6E-06, rx=0.299798, ry=175.773634, rz=18.534319, fatherId=world[0]}
  [685] = {x=-4.7E-05, y=-100.432034, z=-6E-06, rx=0.299796, ry=175.773634, rz=18.534321, fatherId=world[0]}
  [686] = {x=-4.7E-05, y=-100.578931, z=-6E-06, rx=0.299794, ry=175.773634, rz=18.534323, fatherId=world[0]}
  [687] = {x=-4.7E-05, y=-100.725828, z=-6E-06, rx=0.299791, ry=175.773634, rz=18.534326, fatherId=world[0]}
  [688] = {x=-4.7E-05, y=-100.872726, z=-6E-06, rx=0.299789, ry=175.773634, rz=18.534328, fatherId=world[0]}
  [689] = {x=-4.7E-05, y=-101.019623, z=-6E-06, rx=0.299787, ry=175.773634, rz=18.534331, fatherId=world[0]}
  [690] = {x=-4.7E-05, y=-101.16652, z=-6E-06, rx=0.299784, ry=175.773634, rz=18.534333, fatherId=world[0]}
  [691] = {x=-4.7E-05, y=-101.313417, z=-6E-06, rx=0.299782, ry=175.773634, rz=18.534335, fatherId=world[0]}
  [692] = {x=-4.7E-05, y=-101.460314, z=-6E-06, rx=0.29978, ry=175.773634, rz=18.534338, fatherId=world[0]}
  [693] = {x=-4.7E-05, y=-101.607211, z=-6E-06, rx=0.299777, ry=175.773634, rz=18.53434, fatherId=world[0]}
  [694] = {x=-4.7E-05, y=-101.754109, z=-6E-06, rx=0.299775, ry=175.773634, rz=18.534342, fatherId=world[0]}
  [695] = {x=-4.7E-05, y=-101.901006, z=-6E-06, rx=0.299773, ry=175.773635, rz=18.534345, fatherId=world[0]}
  [696] = {x=-4.7E-05, y=-102.047903, z=-6E-06, rx=0.29977, ry=175.773635, rz=18.534347, fatherId=world[0]}
  [697] = {x=-4.7E-05, y=-102.1948, z=-6E-06, rx=0.299768, ry=175.773635, rz=18.534349, fatherId=world[0]}
  [698] = {x=-4.7E-05, y=-102.341697, z=-6E-06, rx=0.299766, ry=175.773635, rz=18.534352, fatherId=world[0]}
  [699] = {x=-4.7E-05, y=-102.488594, z=-6E-06, rx=0.299763, ry=175.773635, rz=18.534354, fatherId=world[0]}
  [700] = {x=-4.7E-05, y=-102.635491, z=-6E-06, rx=0.299761, ry=175.773635, rz=18.534356, fatherId=world[0]}
  [701] = {x=-4.7E-05, y=-102.782389, z=-6E-06, rx=0.299759, ry=175.773635, rz=18.534359, fatherId=world[0]}
  [702] = {x=-4.7E-05, y=-102.929286, z=-6E-06, rx=0.299757, ry=175.773635, rz=18.534361, fatherId=world[0]}
  [703] = {x=-4.7E-05, y=-103.076183, z=-6E-06, rx=0.299754, ry=175.773635, rz=18.534363, fatherId=world[0]}
  [704] = {x=-4.7E-05, y=-103.22308, z=-6E-06, rx=0.299752, ry=175.773635, rz=18.534366, fatherId=world[0]}
  [705] = {x=-4.7E-05, y=-103.369977, z=-6E-06, rx=0.29975, ry=175.773635, rz=18.534368, fatherId=world[0]}
  [706] = {x=-4.8E-05, y=-103.516874, z=-6E-06, rx=0.299747, ry=175.773635, rz=18.53437, fatherId=world[0]}
  [707] = {x=-4.8E-05, y=-103.663771, z=-6E-06, rx=0.299745, ry=175.773635, rz=18.534372, fatherId=world[0]}
  [708] = {x=-4.8E-05, y=-103.810669, z=-6E-06, rx=0.299743, ry=175.773635, rz=18.534375, fatherId=world[0]}
  [709] = {x=-4.8E-05, y=-103.957566, z=-6E-06, rx=0.299741, ry=175.773635, rz=18.534377, fatherId=world[0]}
  [710] = {x=-4.8E-05, y=-104.104463, z=-6E-06, rx=0.299738, ry=175.773636, rz=18.534379, fatherId=world[0]}
  [711] = {x=-4.8E-05, y=-104.25136, z=-6E-06, rx=0.299736, ry=175.773636, rz=18.534382, fatherId=world[0]}
  [712] = {x=-4.8E-05, y=-104.398257, z=-6E-06, rx=0.299734, ry=175.773636, rz=18.534384, fatherId=world[0]}
  [713] = {x=-4.8E-05, y=-104.545154, z=-6E-06, rx=0.299732, ry=175.773636, rz=18.534386, fatherId=world[0]}
  [714] = {x=-4.8E-05, y=-104.692051, z=-6E-06, rx=0.29973, ry=175.773636, rz=18.534388, fatherId=world[0]}
  [715] = {x=-4.8E-05, y=-104.838949, z=-6E-06, rx=0.299727, ry=175.773636, rz=18.534391, fatherId=world[0]}
  [716] = {x=-4.8E-05, y=-104.985846, z=-6E-06, rx=0.299725, ry=175.773636, rz=18.534393, fatherId=world[0]}
  [717] = {x=-4.8E-05, y=-105.132743, z=-6E-06, rx=0.299723, ry=175.773636, rz=18.534395, fatherId=world[0]}
  [718] = {x=-4.8E-05, y=-105.27964, z=-6E-06, rx=0.299721, ry=175.773636, rz=18.534397, fatherId=world[0]}
  [719] = {x=-4.8E-05, y=-105.426537, z=-6E-06, rx=0.299718, ry=175.773636, rz=18.5344, fatherId=world[0]}
  [720] = {x=-4.8E-05, y=-105.573434, z=-6E-06, rx=0.299716, ry=175.773636, rz=18.534402, fatherId=world[0]}
  [721] = {x=-4.8E-05, y=-105.720331, z=-6E-06, rx=0.299714, ry=175.773636, rz=18.534404, fatherId=world[0]}
  [722] = {x=-4.8E-05, y=-105.867229, z=-6E-06, rx=0.299712, ry=175.773636, rz=18.534406, fatherId=world[0]}
  [723] = {x=-4.8E-05, y=-106.014126, z=-6E-06, rx=0.29971, ry=175.773636, rz=18.534408, fatherId=world[0]}
  [724] = {x=-4.8E-05, y=-106.161023, z=-6E-06, rx=0.299707, ry=175.773637, rz=18.534411, fatherId=world[0]}
  [725] = {x=-4.8E-05, y=-106.30792, z=-6E-06, rx=0.299705, ry=175.773637, rz=18.534413, fatherId=world[0]}
  [726] = {x=-4.8E-05, y=-106.454817, z=-6E-06, rx=0.299703, ry=175.773637, rz=18.534415, fatherId=world[0]}
  [727] = {x=-4.8E-05, y=-106.601714, z=-6E-06, rx=0.299701, ry=175.773637, rz=18.534417, fatherId=world[0]}
  [728] = {x=-4.8E-05, y=-106.748611, z=-6E-06, rx=0.299699, ry=175.773637, rz=18.534419, fatherId=world[0]}
  [729] = {x=-4.8E-05, y=-106.895509, z=-6E-06, rx=0.299697, ry=175.773637, rz=18.534422, fatherId=world[0]}
  [730] = {x=-4.8E-05, y=-107.042406, z=-6E-06, rx=0.299694, ry=175.773637, rz=18.534424, fatherId=world[0]}
  [731] = {x=-4.8E-05, y=-107.189303, z=-6E-06, rx=0.299692, ry=175.773637, rz=18.534426, fatherId=world[0]}
  [732] = {x=-4.8E-05, y=-107.3362, z=-6E-06, rx=0.29969, ry=175.773637, rz=18.534428, fatherId=world[0]}
  [733] = {x=-4.8E-05, y=-107.483097, z=-6E-06, rx=0.299688, ry=175.773637, rz=18.53443, fatherId=world[0]}
  [734] = {x=-4.8E-05, y=-107.629994, z=-6E-06, rx=0.299686, ry=175.773637, rz=18.534432, fatherId=world[0]}
  [735] = {x=-4.8E-05, y=-107.776891, z=-6E-06, rx=0.299684, ry=175.773637, rz=18.534435, fatherId=world[0]}
  [736] = {x=-4.8E-05, y=-107.923789, z=-6E-06, rx=0.299682, ry=175.773637, rz=18.534437, fatherId=world[0]}
  [737] = {x=-4.8E-05, y=-108.070686, z=-6E-06, rx=0.299679, ry=175.773638, rz=18.534439, fatherId=world[0]}
  [738] = {x=-4.9E-05, y=-108.217583, z=-6E-06, rx=0.299677, ry=175.773638, rz=18.534441, fatherId=world[0]}
  [739] = {x=-4.9E-05, y=-108.36448, z=-6E-06, rx=0.299675, ry=175.773638, rz=18.534443, fatherId=world[0]}
  [740] = {x=-4.9E-05, y=-108.511377, z=-6E-06, rx=0.299673, ry=175.773638, rz=18.534445, fatherId=world[0]}
  [741] = {x=-4.9E-05, y=-108.658274, z=-6E-06, rx=0.299671, ry=175.773638, rz=18.534448, fatherId=world[0]}
  [742] = {x=-4.9E-05, y=-108.805171, z=-6E-06, rx=0.299669, ry=175.773638, rz=18.53445, fatherId=world[0]}
  [743] = {x=-4.9E-05, y=-108.952069, z=-6E-06, rx=0.299667, ry=175.773638, rz=18.534452, fatherId=world[0]}
  [744] = {x=-4.9E-05, y=-109.098966, z=-6E-06, rx=0.299665, ry=175.773638, rz=18.534454, fatherId=world[0]}
  [745] = {x=-4.9E-05, y=-109.245863, z=-6E-06, rx=0.299663, ry=175.773638, rz=18.534456, fatherId=world[0]}
  [746] = {x=-4.9E-05, y=-109.39276, z=-6E-06, rx=0.29966, ry=175.773638, rz=18.534458, fatherId=world[0]}
  [747] = {x=-4.9E-05, y=-109.539657, z=-6E-06, rx=0.299658, ry=175.773638, rz=18.53446, fatherId=world[0]}
  [748] = {x=-4.9E-05, y=-109.686554, z=-6E-06, rx=0.299656, ry=175.773638, rz=18.534462, fatherId=world[0]}
  [749] = {x=-4.9E-05, y=-109.833452, z=-6E-06, rx=0.299654, ry=175.773639, rz=18.534464, fatherId=world[0]}
  [750] = {x=-4.9E-05, y=-109.980349, z=-6E-06, rx=0.299652, ry=175.773639, rz=18.534467, fatherId=world[0]}
  [751] = {x=-4.9E-05, y=-110.127246, z=-6E-06, rx=0.29965, ry=175.773639, rz=18.534469, fatherId=world[0]}
  [752] = {x=-4.9E-05, y=-110.274143, z=-6E-06, rx=0.299648, ry=175.773639, rz=18.534471, fatherId=world[0]}
  [753] = {x=-4.9E-05, y=-110.42104, z=-6E-06, rx=0.299646, ry=175.773639, rz=18.534473, fatherId=world[0]}
  [754] = {x=-4.9E-05, y=-110.567937, z=-6E-06, rx=0.299644, ry=175.773639, rz=18.534475, fatherId=world[0]}
  [755] = {x=-4.9E-05, y=-110.714834, z=-6E-06, rx=0.299642, ry=175.773639, rz=18.534477, fatherId=world[0]}
  [756] = {x=-4.9E-05, y=-110.861732, z=-6E-06, rx=0.29964, ry=175.773639, rz=18.534479, fatherId=world[0]}
  [757] = {x=-4.9E-05, y=-111.008629, z=-6E-06, rx=0.299638, ry=175.773639, rz=18.534481, fatherId=world[0]}
  [758] = {x=-4.9E-05, y=-111.155526, z=-6E-06, rx=0.299636, ry=175.773639, rz=18.534483, fatherId=world[0]}
  [759] = {x=-4.9E-05, y=-111.302423, z=-6E-06, rx=0.299634, ry=175.773639, rz=18.534485, fatherId=world[0]}
  [760] = {x=-4.9E-05, y=-111.44932, z=-6E-06, rx=0.299632, ry=175.77364, rz=18.534487, fatherId=world[0]}
  [761] = {x=-4.9E-05, y=-111.596217, z=-6E-06, rx=0.29963, ry=175.77364, rz=18.534489, fatherId=world[0]}
  [762] = {x=-4.9E-05, y=-111.743114, z=-6E-06, rx=0.299628, ry=175.77364, rz=18.534491, fatherId=world[0]}
  [763] = {x=-4.9E-05, y=-111.890012, z=-7E-06, rx=0.299626, ry=175.77364, rz=18.534493, fatherId=world[0]}
  [764] = {x=-4.9E-05, y=-112.036909, z=-7E-06, rx=0.299624, ry=175.77364, rz=18.534495, fatherId=world[0]}
  [765] = {x=-4.9E-05, y=-112.183806, z=-7E-06, rx=0.299622, ry=175.77364, rz=18.534497, fatherId=world[0]}
  [766] = {x=-4.9E-05, y=-112.330703, z=-7E-06, rx=0.29962, ry=175.77364, rz=18.534499, fatherId=world[0]}
  [767] = {x=-4.9E-05, y=-112.4776, z=-7E-06, rx=0.299618, ry=175.77364, rz=18.534501, fatherId=world[0]}
  [768] = {x=-4.9E-05, y=-112.624497, z=-7E-06, rx=0.299616, ry=175.77364, rz=18.534504, fatherId=world[0]}
  [769] = {x=-4.9E-05, y=-112.771394, z=-7E-06, rx=0.299614, ry=175.77364, rz=18.534506, fatherId=world[0]}
  [770] = {x=-4.9E-05, y=-112.918292, z=-7E-06, rx=0.299612, ry=175.77364, rz=18.534508, fatherId=world[0]}
  [771] = {x=-4.9E-05, y=-113.065189, z=-7E-06, rx=0.29961, ry=175.773641, rz=18.53451, fatherId=world[0]}
  [772] = {x=-5E-05, y=-113.212086, z=-7E-06, rx=0.299608, ry=175.773641, rz=18.534512, fatherId=world[0]}
  [773] = {x=-5E-05, y=-113.358983, z=-7E-06, rx=0.299606, ry=175.773641, rz=18.534514, fatherId=world[0]}
  [774] = {x=-5E-05, y=-113.50588, z=-7E-06, rx=0.299604, ry=175.773641, rz=18.534515, fatherId=world[0]}
  [775] = {x=-5E-05, y=-113.652777, z=-7E-06, rx=0.299602, ry=175.773641, rz=18.534517, fatherId=world[0]}
  [776] = {x=-5E-05, y=-113.799674, z=-7E-06, rx=0.2996, ry=175.773641, rz=18.534519, fatherId=world[0]}
  [777] = {x=-5E-05, y=-113.946572, z=-7E-06, rx=0.299598, ry=175.773641, rz=18.534521, fatherId=world[0]}
  [778] = {x=-5E-05, y=-114.093469, z=-7E-06, rx=0.299596, ry=175.773641, rz=18.534523, fatherId=world[0]}
  [779] = {x=-5E-05, y=-114.240366, z=-7E-06, rx=0.299594, ry=175.773641, rz=18.534525, fatherId=world[0]}
  [780] = {x=-5E-05, y=-114.387263, z=-7E-06, rx=0.299592, ry=175.773641, rz=18.534527, fatherId=world[0]}
  [781] = {x=-5E-05, y=-114.53416, z=-7E-06, rx=0.29959, ry=175.773641, rz=18.534529, fatherId=world[0]}
  [782] = {x=-5E-05, y=-114.681057, z=-7E-06, rx=0.299588, ry=175.773642, rz=18.534531, fatherId=world[0]}
  [783] = {x=-5E-05, y=-114.827954, z=-7E-06, rx=0.299586, ry=175.773642, rz=18.534533, fatherId=world[0]}
  [784] = {x=-5E-05, y=-114.974852, z=-7E-06, rx=0.299585, ry=175.773642, rz=18.534535, fatherId=world[0]}
  [785] = {x=-5E-05, y=-115.121749, z=-7E-06, rx=0.299583, ry=175.773642, rz=18.534537, fatherId=world[0]}
  [786] = {x=-5E-05, y=-115.268646, z=-7E-06, rx=0.299581, ry=175.773642, rz=18.534539, fatherId=world[0]}
  [787] = {x=-5E-05, y=-115.415543, z=-7E-06, rx=0.299579, ry=175.773642, rz=18.534541, fatherId=world[0]}
  [788] = {x=-5E-05, y=-115.56244, z=-7E-06, rx=0.299577, ry=175.773642, rz=18.534543, fatherId=world[0]}
  [789] = {x=-5E-05, y=-115.709337, z=-7E-06, rx=0.299575, ry=175.773642, rz=18.534545, fatherId=world[0]}
  [790] = {x=-5E-05, y=-115.856235, z=-7E-06, rx=0.299573, ry=175.773642, rz=18.534547, fatherId=world[0]}
  [791] = {x=-5E-05, y=-116.003132, z=-7E-06, rx=0.299571, ry=175.773642, rz=18.534549, fatherId=world[0]}
  [792] = {x=-5E-05, y=-116.150029, z=-7E-06, rx=0.299569, ry=175.773643, rz=18.534551, fatherId=world[0]}
  [793] = {x=-5E-05, y=-116.296926, z=-7E-06, rx=0.299568, ry=175.773643, rz=18.534552, fatherId=world[0]}
  [794] = {x=-5E-05, y=-116.443823, z=-7E-06, rx=0.299566, ry=175.773643, rz=18.534554, fatherId=world[0]}
  [795] = {x=-5E-05, y=-116.59072, z=-7E-06, rx=0.299564, ry=175.773643, rz=18.534556, fatherId=world[0]}
  [796] = {x=-5E-05, y=-116.737617, z=-7E-06, rx=0.299562, ry=175.773643, rz=18.534558, fatherId=world[0]}
  [797] = {x=-5E-05, y=-116.884515, z=-7E-06, rx=0.29956, ry=175.773643, rz=18.53456, fatherId=world[0]}
  [798] = {x=-5E-05, y=-117.031412, z=-7E-06, rx=0.299558, ry=175.773643, rz=18.534562, fatherId=world[0]}
  [799] = {x=-5E-05, y=-117.178309, z=-7E-06, rx=0.299556, ry=175.773643, rz=18.534564, fatherId=world[0]}
  [800] = {x=-5E-05, y=-117.325206, z=-7E-06, rx=0.299555, ry=175.773643, rz=18.534566, fatherId=world[0]}
  [801] = {x=-5E-05, y=-117.472103, z=-7E-06, rx=0.299553, ry=175.773643, rz=18.534567, fatherId=world[0]}
  [802] = {x=-5E-05, y=-117.619, z=-7E-06, rx=0.299551, ry=175.773644, rz=18.534569, fatherId=world[0]}
  [803] = {x=-5E-05, y=-117.765897, z=-7E-06, rx=0.299549, ry=175.773644, rz=18.534571, fatherId=world[0]}
  [804] = {x=-5E-05, y=-117.912795, z=-7E-06, rx=0.299547, ry=175.773644, rz=18.534573, fatherId=world[0]}
  [805] = {x=-5E-05, y=-118.059692, z=-7E-06, rx=0.299545, ry=175.773644, rz=18.534575, fatherId=world[0]}
  [806] = {x=-5E-05, y=-118.206589, z=-7E-06, rx=0.299544, ry=175.773644, rz=18.534577, fatherId=world[0]}
  [807] = {x=-5E-05, y=-118.353486, z=-7E-06, rx=0.299542, ry=175.773644, rz=18.534579, fatherId=world[0]}
  [808] = {x=-5E-05, y=-118.500383, z=-7E-06, rx=0.29954, ry=175.773644, rz=18.53458, fatherId=world[0]}
  [809] = {x=-5E-05, y=-118.64728, z=-7E-06, rx=0.299538, ry=175.773644, rz=18.534582, fatherId=world[0]}
  [810] = {x=-5.1E-05, y=-118.794177, z=-7E-06, rx=0.299536, ry=175.773644, rz=18.534584, fatherId=world[0]}
  [811] = {x=-5.1E-05, y=-118.941075, z=-7E-06, rx=0.299535, ry=175.773645, rz=18.534586, fatherId=world[0]}
  [812] = {x=-5.1E-05, y=-119.087972, z=-7E-06, rx=0.299533, ry=175.773645, rz=18.534588, fatherId=world[0]}
  [813] = {x=-5.1E-05, y=-119.234869, z=-7E-06, rx=0.299531, ry=175.773645, rz=18.53459, fatherId=world[0]}
  [814] = {x=-5.1E-05, y=-119.381766, z=-7E-06, rx=0.299529, ry=175.773645, rz=18.534591, fatherId=world[0]}
  [815] = {x=-5.1E-05, y=-119.528663, z=-7E-06, rx=0.299528, ry=175.773645, rz=18.534593, fatherId=world[0]}
  [816] = {x=-5.1E-05, y=-119.67556, z=-7E-06, rx=0.299526, ry=175.773645, rz=18.534595, fatherId=world[0]}
  [817] = {x=-5.1E-05, y=-119.822457, z=-7E-06, rx=0.299524, ry=175.773645, rz=18.534597, fatherId=world[0]}
  [818] = {x=-5.1E-05, y=-119.969355, z=-7E-06, rx=0.299522, ry=175.773645, rz=18.534599, fatherId=world[0]}
  [819] = {x=-5.1E-05, y=-120.116252, z=-7E-06, rx=0.299521, ry=175.773645, rz=18.5346, fatherId=world[0]}
  [820] = {x=-5.1E-05, y=-120.263149, z=-7E-06, rx=0.299519, ry=175.773646, rz=18.534602, fatherId=world[0]}
  [821] = {x=-5.1E-05, y=-120.410046, z=-7E-06, rx=0.299517, ry=175.773646, rz=18.534604, fatherId=world[0]}
  [822] = {x=-5.1E-05, y=-120.556943, z=-7E-06, rx=0.299515, ry=175.773646, rz=18.534606, fatherId=world[0]}
  [823] = {x=-5.1E-05, y=-120.70384, z=-7E-06, rx=0.299514, ry=175.773646, rz=18.534607, fatherId=world[0]}
  [824] = {x=-5.1E-05, y=-120.850737, z=-7E-06, rx=0.299512, ry=175.773646, rz=18.534609, fatherId=world[0]}
  [825] = {x=-5.1E-05, y=-120.997635, z=-7E-06, rx=0.29951, ry=175.773646, rz=18.534611, fatherId=world[0]}
  [826] = {x=-5.1E-05, y=-121.144532, z=-7E-06, rx=0.299508, ry=175.773646, rz=18.534613, fatherId=world[0]}
  [827] = {x=-5.1E-05, y=-121.291429, z=-7E-06, rx=0.299507, ry=175.773646, rz=18.534614, fatherId=world[0]}
  [828] = {x=-5.1E-05, y=-121.438326, z=-7E-06, rx=0.299505, ry=175.773646, rz=18.534616, fatherId=world[0]}
  [829] = {x=-5.1E-05, y=-121.585223, z=-7E-06, rx=0.299503, ry=175.773647, rz=18.534618, fatherId=world[0]}
  [830] = {x=-5.1E-05, y=-121.73212, z=-7E-06, rx=0.299502, ry=175.773647, rz=18.53462, fatherId=world[0]}
  [831] = {x=-5.1E-05, y=-121.879017, z=-7E-06, rx=0.2995, ry=175.773647, rz=18.534621, fatherId=world[0]}
  [832] = {x=-5.1E-05, y=-122.025915, z=-7E-06, rx=0.299498, ry=175.773647, rz=18.534623, fatherId=world[0]}
  [833] = {x=-5.1E-05, y=-122.172812, z=-7E-06, rx=0.299496, ry=175.773647, rz=18.534625, fatherId=world[0]}
  [834] = {x=-5.1E-05, y=-122.319709, z=-7E-06, rx=0.299495, ry=175.773647, rz=18.534627, fatherId=world[0]}
  [835] = {x=-5.1E-05, y=-122.466606, z=-7E-06, rx=0.299493, ry=175.773647, rz=18.534628, fatherId=world[0]}
  [836] = {x=-5.1E-05, y=-122.613503, z=-7E-06, rx=0.299491, ry=175.773647, rz=18.53463, fatherId=world[0]}
  [837] = {x=-5.1E-05, y=-122.7604, z=-7E-06, rx=0.29949, ry=175.773648, rz=18.534632, fatherId=world[0]}
  [838] = {x=-5.1E-05, y=-122.907298, z=-7E-06, rx=0.299488, ry=175.773648, rz=18.534633, fatherId=world[0]}
  [839] = {x=-5.1E-05, y=-123.054195, z=-7E-06, rx=0.299486, ry=175.773648, rz=18.534635, fatherId=world[0]}
  [840] = {x=-5.1E-05, y=-123.201092, z=-7E-06, rx=0.299485, ry=175.773648, rz=18.534637, fatherId=world[0]}
  [841] = {x=-5.1E-05, y=-123.347989, z=-7E-06, rx=0.299483, ry=175.773648, rz=18.534638, fatherId=world[0]}
  [842] = {x=-5.1E-05, y=-123.494886, z=-7E-06, rx=0.299481, ry=175.773648, rz=18.53464, fatherId=world[0]}
  [843] = {x=-5.1E-05, y=-123.641783, z=-7E-06, rx=0.29948, ry=175.773648, rz=18.534642, fatherId=world[0]}
  [844] = {x=-5.1E-05, y=-123.78868, z=-7E-06, rx=0.299478, ry=175.773648, rz=18.534643, fatherId=world[0]}
  [845] = {x=-5.1E-05, y=-123.935578, z=-8E-06, rx=0.299477, ry=175.773649, rz=18.534645, fatherId=world[0]}
  [846] = {x=-5.1E-05, y=-124.082475, z=-8E-06, rx=0.299475, ry=175.773649, rz=18.534647, fatherId=world[0]}
  [847] = {x=-5.1E-05, y=-124.229372, z=-8E-06, rx=0.299473, ry=175.773649, rz=18.534648, fatherId=world[0]}
  [848] = {x=-5.1E-05, y=-124.376269, z=-8E-06, rx=0.299472, ry=175.773649, rz=18.53465, fatherId=world[0]}
  [849] = {x=-5.1E-05, y=-124.523166, z=-8E-06, rx=0.29947, ry=175.773649, rz=18.534652, fatherId=world[0]}
  [850] = {x=-5.1E-05, y=-124.670063, z=-8E-06, rx=0.299468, ry=175.773649, rz=18.534653, fatherId=world[0]}
  [851] = {x=-5.1E-05, y=-124.81696, z=-8E-06, rx=0.299467, ry=175.773649, rz=18.534655, fatherId=world[0]}
  [852] = {x=-5.1E-05, y=-124.963858, z=-8E-06, rx=0.299465, ry=175.773649, rz=18.534657, fatherId=world[0]}
  [853] = {x=-5.2E-05, y=-125.110755, z=-8E-06, rx=0.299464, ry=175.77365, rz=18.534658, fatherId=world[0]}
  [854] = {x=-5.2E-05, y=-125.257652, z=-8E-06, rx=0.299462, ry=175.77365, rz=18.53466, fatherId=world[0]}
  [855] = {x=-5.2E-05, y=-125.404549, z=-8E-06, rx=0.29946, ry=175.77365, rz=18.534662, fatherId=world[0]}
  [856] = {x=-5.2E-05, y=-125.551446, z=-8E-06, rx=0.299459, ry=175.77365, rz=18.534663, fatherId=world[0]}
  [857] = {x=-5.2E-05, y=-125.698343, z=-8E-06, rx=0.299457, ry=175.77365, rz=18.534665, fatherId=world[0]}
  [858] = {x=-5.2E-05, y=-125.84524, z=-8E-06, rx=0.299456, ry=175.77365, rz=18.534666, fatherId=world[0]}
  [859] = {x=-5.2E-05, y=-125.992138, z=-8E-06, rx=0.299454, ry=175.77365, rz=18.534668, fatherId=world[0]}
  [860] = {x=-5.2E-05, y=-126.139035, z=-8E-06, rx=0.299453, ry=175.77365, rz=18.53467, fatherId=world[0]}
  [861] = {x=-5.2E-05, y=-126.285932, z=-8E-06, rx=0.299451, ry=175.773651, rz=18.534671, fatherId=world[0]}
  [862] = {x=-5.2E-05, y=-126.432829, z=-8E-06, rx=0.299449, ry=175.773651, rz=18.534673, fatherId=world[0]}
  [863] = {x=-5.2E-05, y=-126.579726, z=-8E-06, rx=0.299448, ry=175.773651, rz=18.534674, fatherId=world[0]}
  [864] = {x=-5.2E-05, y=-126.726623, z=-8E-06, rx=0.299446, ry=175.773651, rz=18.534676, fatherId=world[0]}
  [865] = {x=-5.2E-05, y=-126.87352, z=-8E-06, rx=0.299445, ry=175.773651, rz=18.534678, fatherId=world[0]}
  [866] = {x=-5.2E-05, y=-127.020418, z=-8E-06, rx=0.299443, ry=175.773651, rz=18.534679, fatherId=world[0]}
  [867] = {x=-5.2E-05, y=-127.167315, z=-8E-06, rx=0.299442, ry=175.773651, rz=18.534681, fatherId=world[0]}
  [868] = {x=-5.2E-05, y=-127.314212, z=-8E-06, rx=0.29944, ry=175.773651, rz=18.534682, fatherId=world[0]}
  [869] = {x=-5.2E-05, y=-127.461109, z=-8E-06, rx=0.299439, ry=175.773652, rz=18.534684, fatherId=world[0]}
  [870] = {x=-5.2E-05, y=-127.608006, z=-8E-06, rx=0.299437, ry=175.773652, rz=18.534685, fatherId=world[0]}
  [871] = {x=-5.2E-05, y=-127.754903, z=-8E-06, rx=0.299436, ry=175.773652, rz=18.534687, fatherId=world[0]}
  [872] = {x=-5.2E-05, y=-127.9018, z=-8E-06, rx=0.299434, ry=175.773652, rz=18.534689, fatherId=world[0]}
  [873] = {x=-5.2E-05, y=-128.048698, z=-8E-06, rx=0.299433, ry=175.773652, rz=18.53469, fatherId=world[0]}
  [874] = {x=-5.2E-05, y=-128.195595, z=-8E-06, rx=0.299431, ry=175.773652, rz=18.534692, fatherId=world[0]}
  [875] = {x=-5.2E-05, y=-128.342492, z=-8E-06, rx=0.29943, ry=175.773652, rz=18.534693, fatherId=world[0]}
  [876] = {x=-5.2E-05, y=-128.489389, z=-8E-06, rx=0.299428, ry=175.773653, rz=18.534695, fatherId=world[0]}
  [877] = {x=-5.2E-05, y=-128.636286, z=-8E-06, rx=0.299427, ry=175.773653, rz=18.534696, fatherId=world[0]}
  [878] = {x=-5.2E-05, y=-128.783183, z=-8E-06, rx=0.299425, ry=175.773653, rz=18.534698, fatherId=world[0]}
  [879] = {x=-5.2E-05, y=-128.93008, z=-8E-06, rx=0.299424, ry=175.773653, rz=18.534699, fatherId=world[0]}
  [880] = {x=-5.2E-05, y=-129.076978, z=-8E-06, rx=0.299422, ry=175.773653, rz=18.534701, fatherId=world[0]}
  [881] = {x=-5.2E-05, y=-129.223875, z=-8E-06, rx=0.299421, ry=175.773653, rz=18.534702, fatherId=world[0]}
  [882] = {x=-5.2E-05, y=-129.370772, z=-8E-06, rx=0.299419, ry=175.773653, rz=18.534704, fatherId=world[0]}
  [883] = {x=-5.2E-05, y=-129.517669, z=-8E-06, rx=0.299418, ry=175.773653, rz=18.534705, fatherId=world[0]}
  [884] = {x=-5.2E-05, y=-129.664566, z=-8E-06, rx=0.299416, ry=175.773654, rz=18.534707, fatherId=world[0]}
  [885] = {x=-5.2E-05, y=-129.811463, z=-8E-06, rx=0.299415, ry=175.773654, rz=18.534708, fatherId=world[0]}
  [886] = {x=-5.2E-05, y=-129.958361, z=-8E-06, rx=0.299413, ry=175.773654, rz=18.53471, fatherId=world[0]}
  [887] = {x=-5.2E-05, y=-130.105258, z=-8E-06, rx=0.299412, ry=175.773654, rz=18.534711, fatherId=world[0]}
  [888] = {x=-5.2E-05, y=-130.252155, z=-8E-06, rx=0.299411, ry=175.773654, rz=18.534713, fatherId=world[0]}
  [889] = {x=-5.2E-05, y=-130.399052, z=-8E-06, rx=0.299409, ry=175.773654, rz=18.534714, fatherId=world[0]}
  [890] = {x=-5.2E-05, y=-130.545949, z=-8E-06, rx=0.299408, ry=175.773654, rz=18.534716, fatherId=world[0]}
  [891] = {x=-5.2E-05, y=-130.692846, z=-8E-06, rx=0.299406, ry=175.773655, rz=18.534717, fatherId=world[0]}
  [892] = {x=-5.2E-05, y=-130.839743, z=-8E-06, rx=0.299405, ry=175.773655, rz=18.534719, fatherId=world[0]}
  [893] = {x=-5.2E-05, y=-130.986641, z=-8E-06, rx=0.299403, ry=175.773655, rz=18.53472, fatherId=world[0]}
  [894] = {x=-5.2E-05, y=-131.133538, z=-8E-06, rx=0.299402, ry=175.773655, rz=18.534721, fatherId=world[0]}
  [895] = {x=-5.2E-05, y=-131.280435, z=-8E-06, rx=0.299401, ry=175.773655, rz=18.534723, fatherId=world[0]}
  [896] = {x=-5.2E-05, y=-131.427332, z=-8E-06, rx=0.299399, ry=175.773655, rz=18.534724, fatherId=world[0]}
  [897] = {x=-5.2E-05, y=-131.574229, z=-8E-06, rx=0.299398, ry=175.773655, rz=18.534726, fatherId=world[0]}
  [898] = {x=-5.2E-05, y=-131.721126, z=-8E-06, rx=0.299396, ry=175.773656, rz=18.534727, fatherId=world[0]}
  [899] = {x=-5.2E-05, y=-131.868023, z=-8E-06, rx=0.299395, ry=175.773656, rz=18.534729, fatherId=world[0]}
  [900] = {x=-5.2E-05, y=-132.014921, z=-8E-06, rx=0.299394, ry=175.773656, rz=18.53473, fatherId=world[0]}
  [901] = {x=-5.2E-05, y=-132.161818, z=-8E-06, rx=0.299392, ry=175.773656, rz=18.534731, fatherId=world[0]}
  [902] = {x=-5.3E-05, y=-132.308715, z=-8E-06, rx=0.299391, ry=175.773656, rz=18.534733, fatherId=world[0]}
  [903] = {x=-5.3E-05, y=-132.455612, z=-8E-06, rx=0.29939, ry=175.773656, rz=18.534734, fatherId=world[0]}
  [904] = {x=-5.3E-05, y=-132.602509, z=-8E-06, rx=0.299388, ry=175.773656, rz=18.534736, fatherId=world[0]}
  [905] = {x=-5.3E-05, y=-132.749406, z=-8E-06, rx=0.299387, ry=175.773657, rz=18.534737, fatherId=world[0]}
  [906] = {x=-5.3E-05, y=-132.896303, z=-8E-06, rx=0.299385, ry=175.773657, rz=18.534738, fatherId=world[0]}
  [907] = {x=-5.3E-05, y=-133.043201, z=-8E-06, rx=0.299384, ry=175.773657, rz=18.53474, fatherId=world[0]}
  [908] = {x=-5.3E-05, y=-133.190098, z=-8E-06, rx=0.299383, ry=175.773657, rz=18.534741, fatherId=world[0]}
  [909] = {x=-5.3E-05, y=-133.336995, z=-8E-06, rx=0.299381, ry=175.773657, rz=18.534743, fatherId=world[0]}
  [910] = {x=-5.3E-05, y=-133.483892, z=-8E-06, rx=0.29938, ry=175.773657, rz=18.534744, fatherId=world[0]}
  [911] = {x=-5.3E-05, y=-133.630789, z=-8E-06, rx=0.299379, ry=175.773657, rz=18.534745, fatherId=world[0]}
  [912] = {x=-5.3E-05, y=-133.777686, z=-8E-06, rx=0.299377, ry=175.773658, rz=18.534747, fatherId=world[0]}
  [913] = {x=-5.3E-05, y=-133.924583, z=-8E-06, rx=0.299376, ry=175.773658, rz=18.534748, fatherId=world[0]}
  [914] = {x=-5.3E-05, y=-134.071481, z=-8E-06, rx=0.299375, ry=175.773658, rz=18.53475, fatherId=world[0]}
  [915] = {x=-5.3E-05, y=-134.218378, z=-8E-06, rx=0.299373, ry=175.773658, rz=18.534751, fatherId=world[0]}
  [916] = {x=-5.3E-05, y=-134.365275, z=-8E-06, rx=0.299372, ry=175.773658, rz=18.534752, fatherId=world[0]}
  [917] = {x=-5.3E-05, y=-134.512172, z=-8E-06, rx=0.299371, ry=175.773658, rz=18.534754, fatherId=world[0]}
  [918] = {x=-5.3E-05, y=-134.659069, z=-8E-06, rx=0.29937, ry=175.773659, rz=18.534755, fatherId=world[0]}
  [919] = {x=-5.3E-05, y=-134.805966, z=-8E-06, rx=0.299368, ry=175.773659, rz=18.534756, fatherId=world[0]}
  [920] = {x=-5.3E-05, y=-134.952863, z=-8E-06, rx=0.299367, ry=175.773659, rz=18.534758, fatherId=world[0]}
  [921] = {x=-5.3E-05, y=-135.099761, z=-8E-06, rx=0.299366, ry=175.773659, rz=18.534759, fatherId=world[0]}
  [922] = {x=-5.3E-05, y=-135.246658, z=-8E-06, rx=0.299364, ry=175.773659, rz=18.53476, fatherId=world[0]}
  [923] = {x=-5.3E-05, y=-135.393555, z=-9E-06, rx=0.299363, ry=175.773659, rz=18.534762, fatherId=world[0]}
  [924] = {x=-5.3E-05, y=-135.540452, z=-9E-06, rx=0.299362, ry=175.773659, rz=18.534763, fatherId=world[0]}
  [925] = {x=-5.3E-05, y=-135.687349, z=-9E-06, rx=0.299361, ry=175.77366, rz=18.534764, fatherId=world[0]}
  [926] = {x=-5.3E-05, y=-135.834246, z=-9E-06, rx=0.299359, ry=175.77366, rz=18.534765, fatherId=world[0]}
  [927] = {x=-5.3E-05, y=-135.981143, z=-9E-06, rx=0.299358, ry=175.77366, rz=18.534767, fatherId=world[0]}
  [928] = {x=-5.3E-05, y=-136.128041, z=-9E-06, rx=0.299357, ry=175.77366, rz=18.534768, fatherId=world[0]}
  [929] = {x=-5.3E-05, y=-136.274938, z=-9E-06, rx=0.299356, ry=175.77366, rz=18.534769, fatherId=world[0]}
  [930] = {x=-5.3E-05, y=-136.421835, z=-9E-06, rx=0.299354, ry=175.77366, rz=18.534771, fatherId=world[0]}
  [931] = {x=-5.3E-05, y=-136.568732, z=-9E-06, rx=0.299353, ry=175.773661, rz=18.534772, fatherId=world[0]}
  [932] = {x=-5.3E-05, y=-136.715629, z=-9E-06, rx=0.299352, ry=175.773661, rz=18.534773, fatherId=world[0]}
  [933] = {x=-5.3E-05, y=-136.862526, z=-9E-06, rx=0.299351, ry=175.773661, rz=18.534774, fatherId=world[0]}
  [934] = {x=-5.3E-05, y=-137.009424, z=-9E-06, rx=0.299349, ry=175.773661, rz=18.534776, fatherId=world[0]}
  [935] = {x=-5.3E-05, y=-137.156321, z=-9E-06, rx=0.299348, ry=175.773661, rz=18.534777, fatherId=world[0]}
  [936] = {x=-5.3E-05, y=-137.303218, z=-9E-06, rx=0.299347, ry=175.773661, rz=18.534778, fatherId=world[0]}
  [937] = {x=-5.3E-05, y=-137.450115, z=-9E-06, rx=0.299346, ry=175.773662, rz=18.53478, fatherId=world[0]}
  [938] = {x=-5.3E-05, y=-137.597012, z=-9E-06, rx=0.299344, ry=175.773662, rz=18.534781, fatherId=world[0]}
  [939] = {x=-5.3E-05, y=-137.743909, z=-9E-06, rx=0.299343, ry=175.773662, rz=18.534782, fatherId=world[0]}
  [940] = {x=-5.3E-05, y=-137.890806, z=-9E-06, rx=0.299342, ry=175.773662, rz=18.534783, fatherId=world[0]}
  [941] = {x=-5.3E-05, y=-138.037704, z=-9E-06, rx=0.299341, ry=175.773662, rz=18.534785, fatherId=world[0]}
  [942] = {x=-5.3E-05, y=-138.184601, z=-9E-06, rx=0.29934, ry=175.773662, rz=18.534786, fatherId=world[0]}
  [943] = {x=-5.3E-05, y=-138.331498, z=-9E-06, rx=0.299338, ry=175.773662, rz=18.534787, fatherId=world[0]}
  [944] = {x=-5.3E-05, y=-138.478395, z=-9E-06, rx=0.299337, ry=175.773663, rz=18.534788, fatherId=world[0]}
  [945] = {x=-5.3E-05, y=-138.625292, z=-9E-06, rx=0.299336, ry=175.773663, rz=18.534789, fatherId=world[0]}
  [946] = {x=-5.3E-05, y=-138.772189, z=-9E-06, rx=0.299335, ry=175.773663, rz=18.534791, fatherId=world[0]}
  [947] = {x=-5.3E-05, y=-138.919086, z=-9E-06, rx=0.299334, ry=175.773663, rz=18.534792, fatherId=world[0]}
  [948] = {x=-5.3E-05, y=-139.065984, z=-9E-06, rx=0.299333, ry=175.773663, rz=18.534793, fatherId=world[0]}
  [949] = {x=-5.3E-05, y=-139.212881, z=-9E-06, rx=0.299331, ry=175.773663, rz=18.534794, fatherId=world[0]}
  [950] = {x=-5.3E-05, y=-139.359778, z=-9E-06, rx=0.29933, ry=175.773664, rz=18.534795, fatherId=world[0]}
  [951] = {x=-5.3E-05, y=-139.506675, z=-9E-06, rx=0.299329, ry=175.773664, rz=18.534797, fatherId=world[0]}
  [952] = {x=-5.3E-05, y=-139.653572, z=-9E-06, rx=0.299328, ry=175.773664, rz=18.534798, fatherId=world[0]}
  [953] = {x=-5.3E-05, y=-139.800469, z=-9E-06, rx=0.299327, ry=175.773664, rz=18.534799, fatherId=world[0]}
  [954] = {x=-5.3E-05, y=-139.947366, z=-9E-06, rx=0.299326, ry=175.773664, rz=18.5348, fatherId=world[0]}
  [955] = {x=-5.3E-05, y=-140.094264, z=-9E-06, rx=0.299325, ry=175.773664, rz=18.534801, fatherId=world[0]}
  [956] = {x=-5.3E-05, y=-140.241161, z=-9E-06, rx=0.299323, ry=175.773665, rz=18.534803, fatherId=world[0]}
  [957] = {x=-5.3E-05, y=-140.388058, z=-9E-06, rx=0.299322, ry=175.773665, rz=18.534804, fatherId=world[0]}
  [958] = {x=-5.3E-05, y=-140.534955, z=-9E-06, rx=0.299321, ry=175.773665, rz=18.534805, fatherId=world[0]}
  [959] = {x=-5.3E-05, y=-140.681852, z=-9E-06, rx=0.29932, ry=175.773665, rz=18.534806, fatherId=world[0]}
  [960] = {x=-5.3E-05, y=-140.828749, z=-9E-06, rx=0.299319, ry=175.773665, rz=18.534807, fatherId=world[0]}
  [961] = {x=-5.3E-05, y=-140.975646, z=-9E-06, rx=0.299318, ry=175.773665, rz=18.534808, fatherId=world[0]}
  [962] = {x=-5.3E-05, y=-141.122544, z=-9E-06, rx=0.299317, ry=175.773666, rz=18.534809, fatherId=world[0]}
  [963] = {x=-5.3E-05, y=-141.269441, z=-9E-06, rx=0.299316, ry=175.773666, rz=18.534811, fatherId=world[0]}
  [964] = {x=-5.4E-05, y=-141.416338, z=-9E-06, rx=0.299315, ry=175.773666, rz=18.534812, fatherId=world[0]}
  [965] = {x=-5.4E-05, y=-141.563235, z=-9E-06, rx=0.299314, ry=175.773666, rz=18.534813, fatherId=world[0]}
  [966] = {x=-5.4E-05, y=-141.710132, z=-9E-06, rx=0.299312, ry=175.773666, rz=18.534814, fatherId=world[0]}
  [967] = {x=-5.4E-05, y=-141.857029, z=-9E-06, rx=0.299311, ry=175.773666, rz=18.534815, fatherId=world[0]}
  [968] = {x=-5.4E-05, y=-142.003926, z=-9E-06, rx=0.29931, ry=175.773667, rz=18.534816, fatherId=world[0]}
  [969] = {x=-5.4E-05, y=-142.150824, z=-9E-06, rx=0.299309, ry=175.773667, rz=18.534817, fatherId=world[0]}
  [970] = {x=-5.4E-05, y=-142.297721, z=-9E-06, rx=0.299308, ry=175.773667, rz=18.534818, fatherId=world[0]}
  [971] = {x=-5.4E-05, y=-142.444618, z=-9E-06, rx=0.299307, ry=175.773667, rz=18.53482, fatherId=world[0]}
  [972] = {x=-5.4E-05, y=-142.591515, z=-9E-06, rx=0.299306, ry=175.773667, rz=18.534821, fatherId=world[0]}
  [973] = {x=-5.4E-05, y=-142.738412, z=-9E-06, rx=0.299305, ry=175.773668, rz=18.534822, fatherId=world[0]}
  [974] = {x=-5.4E-05, y=-142.885309, z=-9E-06, rx=0.299304, ry=175.773668, rz=18.534823, fatherId=world[0]}
  [975] = {x=-5.4E-05, y=-143.032206, z=-9E-06, rx=0.299303, ry=175.773668, rz=18.534824, fatherId=world[0]}
  [976] = {x=-5.4E-05, y=-143.179104, z=-9E-06, rx=0.299302, ry=175.773668, rz=18.534825, fatherId=world[0]}
  [977] = {x=-5.4E-05, y=-143.326001, z=-9E-06, rx=0.299301, ry=175.773668, rz=18.534826, fatherId=world[0]}
  [978] = {x=-5.4E-05, y=-143.472898, z=-9E-06, rx=0.2993, ry=175.773668, rz=18.534827, fatherId=world[0]}
  [979] = {x=-5.4E-05, y=-143.619795, z=-9E-06, rx=0.299299, ry=175.773669, rz=18.534828, fatherId=world[0]}
  [980] = {x=-5.4E-05, y=-143.766692, z=-9E-06, rx=0.299298, ry=175.773669, rz=18.534829, fatherId=world[0]}
  [981] = {x=-5.4E-05, y=-143.913589, z=-9E-06, rx=0.299297, ry=175.773669, rz=18.53483, fatherId=world[0]}
  [982] = {x=-5.4E-05, y=-144.060487, z=-9E-06, rx=0.299296, ry=175.773669, rz=18.534831, fatherId=world[0]}
  [983] = {x=-5.4E-05, y=-144.207384, z=-9E-06, rx=0.299295, ry=175.773669, rz=18.534832, fatherId=world[0]}
  [984] = {x=-5.4E-05, y=-144.354281, z=-9E-06, rx=0.299294, ry=175.773669, rz=18.534834, fatherId=world[0]}
  [985] = {x=-5.4E-05, y=-144.501178, z=-9E-06, rx=0.299293, ry=175.77367, rz=18.534835, fatherId=world[0]}
  [986] = {x=-5.4E-05, y=-144.648075, z=-9E-06, rx=0.299292, ry=175.77367, rz=18.534836, fatherId=world[0]}
  [987] = {x=-5.4E-05, y=-144.794972, z=-9E-06, rx=0.299291, ry=175.77367, rz=18.534837, fatherId=world[0]}
  [988] = {x=-5.4E-05, y=-144.941869, z=-9E-06, rx=0.29929, ry=175.77367, rz=18.534838, fatherId=world[0]}
  [989] = {x=-5.4E-05, y=-145.088767, z=-9E-06, rx=0.299289, ry=175.77367, rz=18.534839, fatherId=world[0]}
  [990] = {x=-5.4E-05, y=-145.235664, z=-9E-06, rx=0.299288, ry=175.773671, rz=18.53484, fatherId=world[0]}
  [991] = {x=-5.4E-05, y=-145.382561, z=-9E-06, rx=0.299287, ry=175.773671, rz=18.534841, fatherId=world[0]}
